C01839=1169.339,155.960,-56.654,-178.409,6.633,148.750
C01840=1169.335,156.209,-56.676,-178.406,6.635,148.750
C01841=1169.329,156.458,-56.697,-178.404,6.637,148.750
C01842=1169.325,156.707,-56.718,-178.401,6.639,148.749
C01843=1169.321,156.956,-56.739,-178.398,6.640,148.749
C01844=1169.316,157.205,-56.761,-178.396,6.642,148.748
C01845=1169.311,157.454,-56.783,-178.393,6.644,148.748
C01846=1169.306,157.703,-56.803,-178.390,6.646,148.748
C01847=1169.301,157.972,-56.828,-178.388,6.647,148.747
C01848=1169.296,158.241,-56.850,-178.384,6.650,148.747
C01849=1169.290,158.510,-56.874,-178.382,6.652,148.747
C01850=1169.286,158.779,-56.896,-178.378,6.653,148.746
C01851=1169.281,159.028,-56.918,-178.376,6.655,148.746
C01852=1169.276,159.277,-56.940,-178.374,6.657,148.745
C01853=1169.272,159.526,-56.962,-178.370,6.659,148.745
C01854=1169.266,159.775,-56.983,-178.368,6.661,148.745
C01855=1169.262,160.024,-57.005,-178.365,6.663,148.744
C01856=1169.257,160.273,-57.027,-178.362,6.665,148.744
C01857=1169.253,160.522,-57.049,-178.360,6.666,148.744
C01858=1169.248,160.772,-57.070,-178.357,6.668,148.743
C01859=1169.243,161.020,-57.091,-178.354,6.670,148.743
C01860=1169.239,161.270,-57.113,-178.351,6.672,148.742
C01861=1169.234,161.518,-57.135,-178.349,6.673,148.742
C01862=1169.229,161.767,-57.157,-178.346,6.675,148.742
C01863=1169.225,162.016,-57.179,-178.343,6.677,148.741
C01864=1169.220,162.266,-57.200,-178.341,6.679,148.741
C01865=1169.215,162.515,-57.222,-178.338,6.680,148.741
C01866=1169.210,162.764,-57.243,-178.335,6.682,148.740
C01867=1169.206,163.012,-57.265,-178.332,6.685,148.740
C01868=1169.201,163.261,-57.287,-178.329,6.687,148.739
C01869=1169.196,163.510,-57.309,-178.327,6.688,148.739
C01870=1169.192,163.759,-57.331,-178.324,6.690,148.739
C01871=1169.187,164.008,-57.353,-178.322,6.692,148.739
C01872=1169.183,164.257,-57.375,-178.319,6.694,148.738
C01873=1169.178,164.506,-57.396,-178.316,6.696,148.738
C01874=1169.173,164.755,-57.418,-178.314,6.697,148.737
C01875=1169.169,165.004,-57.440,-178.311,6.699,148.737
C01876=1169.164,165.253,-57.462,-178.308,6.701,148.737
C01877=1169.160,165.502,-57.484,-178.306,6.703,148.736
C01878=1169.155,165.751,-57.505,-178.302,6.705,148.736
C01879=1169.150,166.000,-57.528,-178.300,6.707,148.736
C01880=1169.145,166.249,-57.550,-178.297,6.709,148.735
C01881=1169.141,166.498,-57.572,-178.294,6.711,148.735
C01882=1169.136,166.747,-57.593,-178.292,6.712,148.735
C01883=1169.132,166.996,-57.616,-178.289,6.714,148.734
C01884=1169.127,167.245,-57.637,-178.287,6.716,148.734
C01885=1169.123,167.494,-57.659,-178.284,6.718,148.734
C01886=1169.117,167.743,-57.682,-178.281,6.720,148.733
C01887=1169.113,167.993,-57.704,-178.278,6.722,148.733
C01888=1169.108,168.241,-57.725,-178.275,6.724,148.733
C01889=1169.104,168.490,-57.748,-178.273,6.726,148.732
C01890=1169.099,168.739,-57.770,-178.270,6.728,148.732
C01891=1169.094,168.988,-57.792,-178.267,6.729,148.731
C01892=1169.089,169.237,-57.814,-178.265,6.731,148.731
C01893=1169.085,169.486,-57.836,-178.262,6.733,148.731
C01894=1169.080,169.735,-57.858,-178.260,6.735,148.731
C01895=1169.075,169.984,-57.881,-178.257,6.737,148.730
C01896=1169.070,170.233,-57.903,-178.254,6.739,148.730
C01897=1169.066,170.482,-57.925,-178.251,6.741,148.729
C01898=1169.062,170.731,-57.947,-178.248,6.743,148.729
C01899=1169.057,170.980,-57.970,-178.246,6.745,148.729
C01900=1169.052,171.229,-57.992,-178.243,6.746,148.728
C01901=1169.047,171.478,-58.014,-178.240,6.748,148.728
C01902=1169.042,171.727,-58.036,-178.238,6.751,148.728
C01903=1169.038,171.975,-58.059,-178.235,6.753,148.728
C01904=1169.034,172.225,-58.081,-178.232,6.754,148.727
C01905=1169.029,172.474,-58.103,-178.230,6.756,148.727
C01906=1169.024,172.722,-58.126,-178.227,6.758,148.726
C01907=1169.020,172.972,-58.148,-178.224,6.760,148.726
C01908=1169.014,173.221,-58.170,-178.221,6.762,148.726
C01909=1169.010,173.469,-58.193,-178.218,6.764,148.725
C01910=1169.006,173.719,-58.215,-178.216,6.766,148.725
C01911=1169.000,173.968,-58.237,-178.213,6.768,148.725
C01912=1168.996,174.216,-58.260,-178.211,6.770,148.724
C01913=1168.991,174.465,-58.282,-178.208,6.771,148.724
C01914=1168.987,174.714,-58.305,-178.205,6.774,148.724
C01915=1168.983,174.963,-58.327,-178.202,6.776,148.723
C01916=1168.977,175.212,-58.350,-178.199,6.778,148.723
C01917=1168.973,175.461,-58.372,-178.197,6.780,148.723
C01918=1168.968,175.711,-58.395,-178.194,6.781,148.723
C01919=1168.963,175.959,-58.417,-178.192,6.783,148.722
C01920=1168.959,176.208,-58.439,-178.188,6.786,148.722
C01921=1168.954,176.457,-58.463,-178.186,6.788,148.721
C01922=1168.950,176.706,-58.484,-178.183,6.789,148.721
C01923=1168.945,176.955,-58.508,-178.181,6.791,148.721
C01924=1168.941,177.203,-58.530,-178.178,6.793,148.721
C01925=1168.935,177.452,-58.553,-178.176,6.795,148.720
C01926=1168.931,177.701,-58.575,-178.172,6.798,148.720
C01927=1168.926,177.951,-58.598,-178.170,6.799,148.720
C01928=1168.922,178.199,-58.621,-178.167,6.801,148.719
C01929=1168.917,178.448,-58.643,-178.165,6.803,148.719
C01930=1168.913,178.697,-58.666,-178.162,6.805,148.719
C01931=1168.908,178.946,-58.689,-178.159,6.808,148.718
C01932=1168.903,179.195,-58.711,-178.156,6.809,148.718
C01933=1168.898,179.444,-58.734,-178.153,6.811,148.718
C01934=1168.895,179.693,-58.757,-178.151,6.813,148.717
C01935=1168.890,179.942,-58.780,-178.149,6.815,148.717
C01936=1168.885,180.190,-58.802,-178.145,6.818,148.717
C01937=1168.880,180.439,-58.825,-178.143,6.819,148.716
C01938=1168.875,180.689,-58.848,-178.140,6.821,148.716
C01939=1168.871,180.938,-58.871,-178.137,6.823,148.716
C01940=1168.866,181.186,-58.894,-178.134,6.826,148.716
C01941=1168.862,181.435,-58.916,-178.132,6.827,148.715
C01942=1168.857,181.684,-58.939,-178.129,6.829,148.715
C01943=1168.852,181.933,-58.963,-178.126,6.831,148.714
C01944=1168.848,182.182,-58.985,-178.124,6.833,148.714
C01945=1168.843,182.430,-59.008,-178.121,6.836,148.714
C01946=1168.839,182.680,-59.030,-178.118,6.837,148.714
C01947=1168.834,182.929,-59.054,-178.116,6.839,148.713
C01948=1168.829,183.178,-59.077,-178.113,6.841,148.713
C01949=1168.825,183.427,-59.100,-178.110,6.844,148.713
C01950=1168.820,183.675,-59.123,-178.107,6.846,148.712
C01951=1168.815,183.945,-59.148,-178.105,6.847,148.712
C01952=1168.810,184.214,-59.172,-178.101,6.850,148.712
C01953=1168.806,184.485,-59.198,-178.099,6.852,148.711
C01954=1168.800,184.754,-59.223,-178.096,6.854,148.711
C01955=1168.796,185.002,-59.245,-178.093,6.856,148.711
C01956=1168.791,185.251,-59.268,-178.091,6.858,148.711
C01957=1168.786,185.500,-59.292,-178.087,6.861,148.710
C01958=1168.782,185.749,-59.315,-178.085,6.863,148.710
C01959=1168.778,185.998,-59.338,-178.082,6.864,148.710
C01960=1168.773,186.247,-59.361,-178.079,6.866,148.709
C01961=1168.768,186.496,-59.385,-178.077,6.869,148.709
C01962=1168.763,186.745,-59.408,-178.074,6.871,148.709
C01963=1168.759,186.993,-59.430,-178.071,6.873,148.708
C01964=1168.754,187.242,-59.454,-178.069,6.874,148.708
C01965=1168.750,187.491,-59.477,-178.066,6.877,148.708
C01966=1168.745,187.740,-59.501,-178.063,6.879,148.708
C01967=1168.740,187.989,-59.524,-178.060,6.881,148.707
C01968=1168.736,188.238,-59.547,-178.058,6.883,148.707
C01969=1168.731,188.487,-59.570,-178.055,6.886,148.707
C01970=1168.727,188.736,-59.593,-178.052,6.887,148.706
C01971=1168.722,188.985,-59.617,-178.050,6.889,148.706
C01972=1168.717,189.234,-59.640,-178.047,6.891,148.706
C01973=1168.712,189.483,-59.663,-178.044,6.894,148.706
C01974=1168.707,189.732,-59.686,-178.041,6.896,148.705
C01975=1168.704,189.980,-59.710,-178.039,6.897,148.705
C01976=1168.699,190.229,-59.733,-178.036,6.900,148.705
C01977=1168.694,190.478,-59.757,-178.033,6.902,148.704
C01978=1168.690,190.727,-59.780,-178.031,6.904,148.704
C01979=1168.685,190.976,-59.803,-178.028,6.906,148.704
C01980=1168.680,191.225,-59.827,-178.025,6.909,148.704
C01981=1168.676,191.473,-59.851,-178.023,6.910,148.703
C01982=1168.671,191.722,-59.874,-178.020,6.912,148.703
C01983=1168.666,191.971,-59.897,-178.017,6.915,148.703
C01984=1168.662,192.220,-59.921,-178.014,6.917,148.702
C01985=1168.657,192.469,-59.945,-178.012,6.919,148.702
C01986=1168.653,192.718,-59.968,-178.009,6.920,148.702
C01987=1168.648,192.967,-59.992,-178.006,6.923,148.702
C01988=1168.643,193.216,-60.015,-178.004,6.925,148.701
C01989=1168.639,193.464,-60.039,-178.001,6.927,148.701
C01990=1168.634,193.713,-60.062,-177.998,6.929,148.701
C01991=1168.629,193.962,-60.086,-177.995,6.932,148.700
C01992=1168.625,194.211,-60.110,-177.993,6.933,148.700
C01993=1168.620,194.460,-60.133,-177.990,6.936,148.700
C01994=1168.616,194.709,-60.157,-177.987,6.938,148.700
C01995=1168.611,194.957,-60.181,-177.985,6.940,148.699
C01996=1168.607,195.206,-60.204,-177.981,6.942,148.699
C01997=1168.602,195.455,-60.228,-177.979,6.945,148.699
C01998=1168.597,195.704,-60.251,-177.977,6.946,148.698
C01999=1168.593,195.953,-60.275,-177.974,6.948,148.698
C02000=1168.588,196.201,-60.299,-177.971,6.951,148.698
C02001=1168.584,196.450,-60.322,-177.968,6.953,148.698
C02002=1168.579,196.699,-60.346,-177.966,6.955,148.697
C02003=1168.575,196.948,-60.370,-177.963,6.957,148.697
C02004=1168.571,197.197,-60.394,-177.960,6.959,148.697
C02005=1168.566,197.446,-60.417,-177.958,6.961,148.696
C02006=1168.561,197.695,-60.442,-177.955,6.964,148.696
C02007=1168.556,197.944,-60.466,-177.952,6.966,148.696
C02008=1168.552,198.192,-60.490,-177.950,6.968,148.696
C02009=1168.547,198.441,-60.513,-177.947,6.970,148.696
C02010=1168.543,198.689,-60.537,-177.944,6.972,148.695
C02011=1168.538,198.938,-60.560,-177.941,6.974,148.695
C02012=1168.534,199.187,-60.584,-177.939,6.977,148.695
C02013=1168.529,199.436,-60.609,-177.936,6.979,148.694
C02014=1168.524,199.685,-60.633,-177.933,6.981,148.694
C02015=1168.520,199.934,-60.657,-177.930,6.983,148.694
C02016=1168.515,200.183,-60.680,-177.928,6.985,148.694
C02017=1168.511,200.431,-60.704,-177.925,6.988,148.693
C02018=1168.507,200.680,-60.728,-177.922,6.990,148.693
C02019=1168.501,200.929,-60.752,-177.920,6.992,148.693
C02020=1168.497,201.178,-60.777,-177.916,6.994,148.692
C02021=1168.493,201.426,-60.801,-177.914,6.996,148.692
C02022=1168.488,201.675,-60.824,-177.912,6.998,148.692
C02023=1168.483,201.924,-60.849,-177.908,7.001,148.692
C02024=1168.479,202.173,-60.873,-177.906,7.003,148.692
C02025=1168.474,202.421,-60.897,-177.903,7.005,148.691
C02026=1168.470,202.671,-60.921,-177.901,7.008,148.691
C02027=1168.465,202.919,-60.945,-177.898,7.009,148.691
C02028=1168.461,203.168,-60.970,-177.895,7.012,148.690
C02029=1168.456,203.416,-60.994,-177.893,7.014,148.690
C02030=1168.451,203.666,-61.018,-177.890,7.016,148.690
C02031=1168.447,203.915,-61.042,-177.887,7.018,148.690
C02032=1168.443,204.163,-61.066,-177.884,7.021,148.690
C02033=1168.438,204.412,-61.091,-177.882,7.022,148.689
C02034=1168.433,204.660,-61.115,-177.879,7.025,148.689
C02035=1168.429,204.909,-61.139,-177.876,7.027,148.689
C02036=1168.424,205.159,-61.163,-177.873,7.030,148.688
C02037=1168.419,205.407,-61.187,-177.871,7.032,148.688
C02038=1168.415,205.656,-61.211,-177.868,7.034,148.688
C02039=1168.411,205.905,-61.236,-177.865,7.037,148.688
C02040=1168.406,206.153,-61.260,-177.863,7.038,148.688
C02041=1168.401,206.402,-61.285,-177.860,7.041,148.687
C02042=1168.397,206.651,-61.309,-177.857,7.043,148.687
C02043=1168.393,206.900,-61.334,-177.855,7.045,148.687
C02044=1168.388,207.148,-61.358,-177.852,7.048,148.687
C02045=1168.383,207.397,-61.382,-177.849,7.050,148.686
C02046=1168.379,207.646,-61.407,-177.846,7.052,148.686
C02047=1168.374,207.895,-61.432,-177.844,7.054,148.686
C02048=1168.369,208.143,-61.456,-177.841,7.056,148.686
C02049=1168.365,208.392,-61.480,-177.838,7.059,148.685
C02050=1168.360,208.641,-61.505,-177.836,7.061,148.685
C02051=1168.356,208.890,-61.529,-177.832,7.063,148.685
C02052=1168.351,209.138,-61.554,-177.830,7.065,148.685
C02053=1168.347,209.387,-61.578,-177.827,7.068,148.684
C02054=1168.342,209.636,-61.603,-177.825,7.070,148.684
C02055=1168.337,209.906,-61.629,-177.822,7.073,148.684
C02056=1168.333,210.177,-61.656,-177.819,7.075,148.684
C02057=1168.328,210.447,-61.683,-177.816,7.078,148.683
C02058=1168.323,210.717,-61.710,-177.813,7.080,148.683
C02059=1168.318,210.967,-61.735,-177.810,7.082,148.683
C02060=1168.314,211.215,-61.759,-177.807,7.085,148.683
C02061=1168.309,211.465,-61.784,-177.805,7.087,148.682
C02062=1168.304,211.713,-61.809,-177.802,7.090,148.682
C02063=1168.300,211.962,-61.833,-177.799,7.091,148.682
C02064=1168.295,212.210,-61.858,-177.797,7.094,148.682
C02065=1168.291,212.459,-61.882,-177.794,7.096,148.681
C02066=1168.286,212.708,-61.908,-177.792,7.098,148.681
C02067=1168.281,212.957,-61.932,-177.788,7.101,148.681
C02068=1168.277,213.205,-61.957,-177.786,7.103,148.681
C02069=1168.273,213.454,-61.982,-177.783,7.106,148.681
C02070=1168.268,213.703,-62.006,-177.780,7.107,148.680
C02071=1168.264,213.952,-62.031,-177.778,7.110,148.680
C02072=1168.259,214.200,-62.057,-177.775,7.112,148.680
C02073=1168.255,214.449,-62.081,-177.773,7.114,148.680
C02074=1168.250,214.698,-62.106,-177.769,7.117,148.679
C02075=1168.245,214.946,-62.131,-177.767,7.119,148.679
C02076=1168.241,215.195,-62.155,-177.764,7.122,148.679
C02077=1168.236,215.444,-62.180,-177.762,7.124,148.679
C02078=1168.232,215.693,-62.206,-177.759,7.126,148.679
C02079=1168.228,215.941,-62.230,-177.756,7.128,148.678
C02080=1168.223,216.190,-62.256,-177.753,7.131,148.678
C02081=1168.218,216.439,-62.280,-177.751,7.133,148.678
C02082=1168.214,216.688,-62.305,-177.748,7.136,148.678
C02083=1168.210,216.936,-62.330,-177.746,7.138,148.678
C02084=1168.205,217.185,-62.355,-177.742,7.140,148.677
C02085=1168.200,217.433,-62.381,-177.740,7.143,148.677
C02086=1168.195,217.682,-62.405,-177.737,7.145,148.677
C02087=1168.192,217.931,-62.430,-177.735,7.147,148.677
C02088=1168.187,218.179,-62.455,-177.731,7.150,148.676
C02089=1168.182,218.428,-62.481,-177.729,7.152,148.676
C02090=1168.178,218.678,-62.506,-177.727,7.154,148.676
C02091=1168.173,218.926,-62.531,-177.724,7.157,148.676
C02092=1168.169,219.175,-62.556,-177.721,7.159,148.676
C02093=1168.164,219.423,-62.581,-177.718,7.161,148.675
C02094=1168.160,219.672,-62.607,-177.716,7.163,148.675
C02095=1168.155,219.920,-62.632,-177.713,7.166,148.675
C02096=1168.151,220.169,-62.657,-177.710,7.168,148.675
C02097=1168.146,220.418,-62.681,-177.708,7.171,148.675
C02098=1168.142,220.666,-62.707,-177.705,7.173,148.674
C02099=1168.137,220.915,-62.732,-177.702,7.176,148.674
C02100=1168.133,221.164,-62.758,-177.699,7.177,148.674
C02101=1168.129,221.413,-62.783,-177.697,7.180,148.674
C02102=1168.124,221.661,-62.809,-177.694,7.182,148.673
C02103=1168.119,221.910,-62.834,-177.691,7.185,148.673
C02104=1168.114,222.158,-62.859,-177.688,7.188,148.673
C02105=1168.110,222.407,-62.885,-177.686,7.190,148.673
C02106=1168.106,222.656,-62.909,-177.683,7.193,148.673
C02107=1168.102,222.904,-62.935,-177.680,7.195,148.673
C02108=1168.097,223.153,-62.960,-177.678,7.198,148.672
C02109=1168.093,223.401,-62.986,-177.675,7.199,148.672
C02110=1168.088,223.651,-63.011,-177.672,7.202,148.672
C02111=1168.084,223.900,-63.037,-177.670,7.204,148.672
C02112=1168.079,224.148,-63.062,-177.667,7.207,148.672
C02113=1168.075,224.397,-63.088,-177.664,7.209,148.671
C02114=1168.070,224.645,-63.113,-177.661,7.212,148.671
C02115=1168.065,224.894,-63.138,-177.659,7.214,148.671
C02116=1168.061,225.143,-63.164,-177.656,7.217,148.671
C02117=1168.056,225.391,-63.189,-177.654,7.219,148.671
C02118=1168.052,225.640,-63.215,-177.650,7.221,148.670
C02119=1168.048,225.889,-63.241,-177.648,7.223,148.670
C02120=1168.043,226.137,-63.266,-177.645,7.226,148.670
C02121=1168.039,226.385,-63.292,-177.642,7.229,148.670
C02122=1168.035,226.634,-63.318,-177.640,7.231,148.670
C02123=1168.030,226.882,-63.343,-177.637,7.234,148.669
C02124=1168.025,227.132,-63.369,-177.635,7.236,148.669
C02125=1168.020,227.381,-63.394,-177.631,7.238,148.669
C02126=1168.015,227.629,-63.420,-177.629,7.241,148.669
C02127=1168.011,227.878,-63.446,-177.626,7.243,148.669
C02128=1168.007,228.127,-63.471,-177.624,7.245,148.669
C02129=1168.003,228.375,-63.497,-177.621,7.248,148.668
C02130=1167.998,228.624,-63.522,-177.618,7.251,148.668
C02131=1167.994,228.872,-63.548,-177.616,7.253,148.668
C02132=1167.990,229.121,-63.574,-177.612,7.256,148.668
C02133=1167.985,229.370,-63.601,-177.610,7.258,148.668
C02134=1167.980,229.618,-63.626,-177.607,7.261,148.668
C02135=1167.976,229.867,-63.652,-177.605,7.262,148.667
C02136=1167.972,230.115,-63.678,-177.602,7.265,148.667
C02137=1167.967,230.364,-63.704,-177.599,7.268,148.667
C02138=1167.963,230.612,-63.729,-177.597,7.270,148.667
C02139=1167.958,230.861,-63.755,-177.594,7.273,148.667
C02140=1167.953,231.110,-63.781,-177.591,7.275,148.666
C02141=1167.949,231.359,-63.807,-177.588,7.278,148.666
C02142=1167.945,231.606,-63.833,-177.586,7.280,148.666
C02143=1167.940,231.856,-63.859,-177.583,7.283,148.666
C02144=1167.935,232.104,-63.885,-177.580,7.286,148.666
C02145=1167.931,232.353,-63.911,-177.578,7.287,148.665
C02146=1167.927,232.602,-63.937,-177.575,7.290,148.665
C02147=1167.922,232.850,-63.963,-177.573,7.292,148.665
C02148=1167.917,233.099,-63.989,-177.569,7.295,148.665
C02149=1167.913,233.347,-64.015,-177.567,7.298,148.665
C02150=1167.909,233.596,-64.041,-177.564,7.300,148.665
C02151=1167.904,233.845,-64.068,-177.561,7.303,148.664
C02152=1167.900,234.093,-64.093,-177.559,7.305,148.664
C02153=1167.895,234.342,-64.119,-177.556,7.308,148.664
C02154=1167.891,234.590,-64.146,-177.553,7.310,148.664
C02155=1167.886,234.839,-64.172,-177.551,7.313,148.664
C02156=1167.882,235.088,-64.197,-177.548,7.316,148.664
C02157=1167.878,235.336,-64.224,-177.545,7.317,148.663
C02158=1167.873,235.585,-64.250,-177.543,7.320,148.663
C02159=1167.868,235.856,-64.278,-177.539,7.323,148.663
C02160=1167.863,236.128,-64.307,-177.537,7.326,148.663
C02161=1167.859,236.399,-64.336,-177.534,7.329,148.663
C02162=1167.853,236.671,-64.365,-177.531,7.331,148.663
C02163=1167.849,236.919,-64.391,-177.528,7.334,148.663
C02164=1167.845,237.168,-64.417,-177.526,7.336,148.663
C02165=1167.840,237.417,-64.444,-177.523,7.339,148.662
C02166=1167.836,237.666,-64.470,-177.520,7.341,148.662
C02167=1167.831,237.914,-64.497,-177.518,7.344,148.662
C02168=1167.827,238.163,-64.522,-177.514,7.347,148.662
C02169=1167.823,238.411,-64.549,-177.512,7.349,148.662
C02170=1167.818,238.660,-64.575,-177.509,7.352,148.662
C02171=1167.814,238.908,-64.601,-177.506,7.355,148.661
C02172=1167.809,239.157,-64.628,-177.504,7.357,148.661
C02173=1167.805,239.405,-64.654,-177.501,7.360,148.661
C02174=1167.800,239.654,-64.680,-177.498,7.363,148.661
C02175=1167.796,239.902,-64.707,-177.496,7.364,148.661
C02176=1167.791,240.151,-64.734,-177.493,7.367,148.661
C02177=1167.787,240.400,-64.760,-177.490,7.370,148.661
C02178=1167.782,240.648,-64.787,-177.488,7.372,148.660
C02179=1167.778,240.897,-64.813,-177.485,7.375,148.660
C02180=1167.774,241.145,-64.840,-177.483,7.377,148.660
C02181=1167.769,241.394,-64.867,-177.480,7.380,148.660
C02182=1167.765,241.643,-64.892,-177.477,7.383,148.660
C02183=1167.760,241.891,-64.919,-177.474,7.385,148.660
C02184=1167.756,242.139,-64.946,-177.472,7.388,148.660
C02185=1167.752,242.388,-64.973,-177.469,7.391,148.659
C02186=1167.747,242.637,-64.999,-177.466,7.393,148.659
C02187=1167.743,242.885,-65.026,-177.464,7.395,148.659
C02188=1167.738,243.134,-65.053,-177.461,7.398,148.659
C02189=1167.734,243.382,-65.079,-177.459,7.401,148.659
C02190=1167.729,243.631,-65.106,-177.455,7.403,148.659
C02191=1167.725,243.879,-65.132,-177.453,7.406,148.659
C02192=1167.721,244.128,-65.159,-177.450,7.409,148.658
C02193=1167.716,244.376,-65.186,-177.448,7.411,148.658
C02194=1167.712,244.624,-65.213,-177.444,7.414,148.658
C02195=1167.707,244.873,-65.239,-177.442,7.417,148.658
C02196=1167.702,245.122,-65.266,-177.440,7.419,148.658
C02197=1167.698,245.370,-65.293,-177.437,7.422,148.658
C02198=1167.694,245.619,-65.320,-177.434,7.425,148.658
C02199=1167.690,245.868,-65.347,-177.431,7.427,148.657
C02200=1167.685,246.116,-65.374,-177.429,7.430,148.657
C02201=1167.681,246.364,-65.401,-177.426,7.433,148.657
C02202=1167.676,246.613,-65.428,-177.424,7.435,148.657
C02203=1167.672,246.861,-65.455,-177.420,7.437,148.657
C02204=1167.668,247.110,-65.481,-177.418,7.440,148.657
C02205=1167.663,247.358,-65.508,-177.415,7.442,148.657
C02206=1167.659,247.607,-65.535,-177.413,7.445,148.657
C02207=1167.654,247.855,-65.562,-177.410,7.448,148.657
C02208=1167.650,248.103,-65.589,-177.407,7.451,148.656
C02209=1167.646,248.353,-65.616,-177.405,7.453,148.656
C02210=1167.641,248.601,-65.643,-177.402,7.456,148.656
C02211=1167.637,248.850,-65.670,-177.399,7.459,148.656
C02212=1167.632,249.098,-65.697,-177.397,7.461,148.656
C02213=1167.628,249.346,-65.724,-177.394,7.464,148.656
C02214=1167.623,249.595,-65.751,-177.391,7.467,148.656
C02215=1167.619,249.843,-65.778,-177.388,7.470,148.656
C02216=1167.615,250.092,-65.805,-177.386,7.472,148.656
C02217=1167.610,250.341,-65.833,-177.383,7.475,148.655
C02218=1167.605,250.589,-65.860,-177.380,7.478,148.655
C02219=1167.601,250.838,-65.887,-177.378,7.480,148.655
C02220=1167.597,251.085,-65.914,-177.375,7.482,148.655
C02221=1167.593,251.335,-65.941,-177.372,7.485,148.655
C02222=1167.588,251.583,-65.968,-177.369,7.488,148.655
C02223=1167.584,251.832,-65.995,-177.367,7.491,148.655
C02224=1167.579,252.080,-66.022,-177.365,7.493,148.655
C02225=1167.575,252.328,-66.050,-177.362,7.496,148.655
C02226=1167.571,252.577,-66.078,-177.359,7.499,148.654
C02227=1167.566,252.826,-66.105,-177.356,7.501,148.654
C02228=1167.561,253.074,-66.132,-177.354,7.504,148.654
C02229=1167.557,253.322,-66.160,-177.351,7.507,148.654
C02230=1167.552,253.571,-66.187,-177.348,7.510,148.654
C02231=1167.548,253.820,-66.214,-177.346,7.512,148.654
C02232=1167.544,254.068,-66.242,-177.343,7.515,148.654
C02233=1167.540,254.316,-66.268,-177.340,7.518,148.654
C02234=1167.535,254.564,-66.295,-177.337,7.521,148.654
C02235=1167.532,254.813,-66.323,-177.335,7.523,148.654
C02236=1167.527,255.061,-66.351,-177.332,7.526,148.653
C02237=1167.522,255.310,-66.378,-177.330,7.529,148.653
C02238=1167.517,255.558,-66.406,-177.327,7.532,148.653
C02239=1167.513,255.807,-66.433,-177.325,7.534,148.653
C02240=1167.509,256.055,-66.461,-177.322,7.537,148.653
C02241=1167.504,256.304,-66.488,-177.319,7.540,148.653
C02242=1167.500,256.552,-66.516,-177.316,7.542,148.653
C02243=1167.496,256.801,-66.543,-177.314,7.545,148.653
C02244=1167.491,257.049,-66.571,-177.311,7.548,148.653
C02245=1167.487,257.298,-66.599,-177.308,7.551,148.653
C02246=1167.483,257.546,-66.626,-177.305,7.553,148.653
C02247=1167.478,257.794,-66.653,-177.303,7.556,148.652
C02248=1167.474,258.043,-66.681,-177.300,7.559,148.652
C02249=1167.470,258.291,-66.709,-177.298,7.562,148.652
C02250=1167.465,258.539,-66.737,-177.295,7.564,148.652
C02251=1167.461,258.789,-66.765,-177.292,7.567,148.652
C02252=1167.456,259.036,-66.792,-177.290,7.570,148.652
C02253=1167.452,259.285,-66.819,-177.287,7.572,148.652
C02254=1167.448,259.534,-66.847,-177.284,7.575,148.652
C02255=1167.444,259.781,-66.875,-177.281,7.578,148.652
C02256=1167.439,260.030,-66.902,-177.279,7.580,148.652
C02257=1167.435,260.279,-66.931,-177.276,7.583,148.652
C02258=1167.430,260.527,-66.958,-177.274,7.586,148.652
C02259=1167.426,260.775,-66.986,-177.271,7.589,148.651
C02260=1167.422,261.024,-67.014,-177.268,7.592,148.651
C02261=1167.417,261.272,-67.042,-177.266,7.594,148.651
C02262=1167.413,261.521,-67.070,-177.263,7.597,148.651
C02263=1167.407,261.794,-67.100,-177.260,7.600,148.651
C02264=1167.403,262.067,-67.131,-177.257,7.604,148.651
C02265=1167.398,262.340,-67.162,-177.254,7.607,148.651
C02266=1167.394,262.613,-67.193,-177.251,7.610,148.651
C02267=1167.389,262.862,-67.220,-177.248,7.612,148.651
C02268=1167.385,263.110,-67.248,-177.246,7.615,148.651
C02269=1167.380,263.358,-67.276,-177.243,7.618,148.651
C02270=1167.376,263.606,-67.304,-177.241,7.621,148.651
C02271=1167.372,263.855,-67.332,-177.238,7.624,148.651
C02272=1167.367,264.104,-67.360,-177.235,7.626,148.651
C02273=1167.363,264.352,-67.388,-177.232,7.629,148.650
C02274=1167.359,264.600,-67.416,-177.230,7.632,148.650
C02275=1167.354,264.849,-67.445,-177.227,7.635,148.650
C02276=1167.350,265.097,-67.472,-177.225,7.638,148.650
C02277=1167.346,265.345,-67.501,-177.222,7.640,148.650
C02278=1167.341,265.594,-67.529,-177.219,7.643,148.650
C02279=1167.337,265.842,-67.557,-177.217,7.646,148.650
C02280=1167.333,266.090,-67.585,-177.214,7.649,148.650
C02281=1167.328,266.339,-67.614,-177.212,7.651,148.650
C02282=1167.324,266.587,-67.641,-177.209,7.654,148.650
C02283=1167.319,266.836,-67.670,-177.206,7.657,148.650
C02284=1167.315,267.084,-67.698,-177.203,7.660,148.650
C02285=1167.311,267.332,-67.726,-177.201,7.663,148.650
C02286=1167.306,267.580,-67.754,-177.198,7.665,148.650
C02287=1167.303,267.829,-67.783,-177.196,7.668,148.650
C02288=1167.297,268.077,-67.811,-177.193,7.671,148.650
C02289=1167.294,268.326,-67.839,-177.190,7.674,148.650
C02290=1167.289,268.574,-67.867,-177.187,7.677,148.649
C02291=1167.285,268.822,-67.896,-177.185,7.679,148.649
C02292=1167.280,269.071,-67.924,-177.182,7.682,148.649
C02293=1167.276,269.319,-67.952,-177.180,7.686,148.650
C02294=1167.272,269.568,-67.981,-177.177,7.689,148.649
C02295=1167.267,269.816,-68.009,-177.175,7.692,148.649
C02296=1167.263,270.065,-68.037,-177.172,7.695,148.649
C02297=1167.259,270.312,-68.066,-177.169,7.698,148.649
C02298=1167.254,270.561,-68.095,-177.167,7.700,148.649
C02299=1167.250,270.809,-68.122,-177.164,7.703,148.649
C02300=1167.245,271.058,-68.151,-177.161,7.706,148.649
C02301=1167.242,271.306,-68.179,-177.159,7.709,148.649
C02302=1167.237,271.554,-68.208,-177.156,7.712,148.649
C02303=1167.232,271.803,-68.237,-177.153,7.715,148.649
C02304=1167.228,272.051,-68.265,-177.150,7.717,148.649
C02305=1167.223,272.300,-68.294,-177.148,7.720,148.649
C02306=1167.220,272.548,-68.322,-177.145,7.723,148.649
C02307=1167.215,272.796,-68.351,-177.143,7.726,148.649
C02308=1167.210,273.045,-68.380,-177.140,7.729,148.649
C02309=1167.207,273.293,-68.408,-177.138,7.732,148.649
C02310=1167.202,273.541,-68.437,-177.135,7.735,148.649
C02311=1167.197,273.790,-68.466,-177.132,7.738,148.649
C02312=1167.194,274.038,-68.494,-177.130,7.740,148.649
C02313=1167.189,274.286,-68.523,-177.127,7.743,148.649
C02314=1167.185,274.534,-68.552,-177.124,7.746,148.649
C02315=1167.181,274.783,-68.580,-177.122,7.749,148.649
C02316=1167.176,275.031,-68.609,-177.119,7.752,148.649
C02317=1167.172,275.279,-68.638,-177.116,7.755,148.648
C02318=1167.168,275.528,-68.666,-177.113,7.758,148.648
C02319=1167.163,275.775,-68.695,-177.111,7.761,148.649
C02320=1167.159,276.024,-68.724,-177.109,7.763,148.648
C02321=1167.155,276.272,-68.753,-177.106,7.766,148.648
C02322=1167.151,276.521,-68.782,-177.104,7.769,148.648
C02323=1167.146,276.769,-68.811,-177.101,7.772,148.648
C02324=1167.141,277.017,-68.840,-177.098,7.775,148.648
C02325=1167.138,277.265,-68.868,-177.095,7.778,148.648
C02326=1167.133,277.514,-68.897,-177.093,7.781,148.648
C02327=1167.129,277.762,-68.926,-177.090,7.784,148.648
C02328=1167.124,278.011,-68.955,-177.087,7.787,148.648
C02329=1167.120,278.259,-68.984,-177.085,7.789,148.648
C02330=1167.116,278.506,-69.013,-177.083,7.792,148.648
C02331=1167.112,278.755,-69.042,-177.080,7.795,148.648
C02332=1167.107,279.003,-69.071,-177.077,7.798,148.648
C02333=1167.103,279.252,-69.101,-177.074,7.801,148.648
C02334=1167.099,279.501,-69.129,-177.072,7.804,148.648
C02335=1167.095,279.748,-69.158,-177.069,7.807,148.648
C02336=1167.090,279.996,-69.187,-177.067,7.810,148.648
C02337=1167.086,280.245,-69.216,-177.064,7.813,148.648
C02338=1167.082,280.493,-69.245,-177.061,7.816,148.648
C02339=1167.078,280.741,-69.275,-177.058,7.819,148.648
C02340=1167.073,280.990,-69.303,-177.056,7.821,148.648
C02341=1167.068,281.238,-69.333,-177.054,7.825,148.648
C02342=1167.064,281.486,-69.362,-177.051,7.828,148.648
C02343=1167.060,281.734,-69.392,-177.048,7.831,148.648
C02344=1167.056,281.983,-69.421,-177.046,7.834,148.648
C02345=1167.051,282.231,-69.449,-177.043,7.837,148.648
C02346=1167.047,282.479,-69.478,-177.040,7.840,148.648
C02347=1167.043,282.727,-69.508,-177.038,7.843,148.648
C02348=1167.039,282.975,-69.537,-177.035,7.846,148.648
C02349=1167.035,283.224,-69.567,-177.032,7.849,148.648
C02350=1167.031,283.472,-69.596,-177.030,7.852,148.648
C02351=1167.025,283.720,-69.625,-177.027,7.855,148.648
C02352=1167.021,283.968,-69.654,-177.024,7.858,148.648
C02353=1167.017,284.217,-69.683,-177.022,7.860,148.648
C02354=1167.013,284.465,-69.713,-177.020,7.863,148.648
C02355=1167.009,284.713,-69.742,-177.017,7.866,148.648
C02356=1167.005,284.961,-69.772,-177.014,7.869,148.648
C02357=1167.000,285.210,-69.801,-177.012,7.872,148.648
C02358=1166.996,285.458,-69.831,-177.009,7.875,148.648
C02359=1166.991,285.707,-69.861,-177.006,7.878,148.648
C02360=1166.986,285.954,-69.890,-177.004,7.881,148.648
C02361=1166.982,286.202,-69.919,-177.001,7.885,148.648
C02362=1166.978,286.451,-69.949,-176.998,7.887,148.648
C02363=1166.974,286.699,-69.978,-176.996,7.890,148.648
C02364=1166.970,286.947,-70.008,-176.993,7.893,148.648
C02365=1166.966,287.196,-70.037,-176.990,7.896,148.648
C02366=1166.961,287.444,-70.067,-176.988,7.900,148.648
C02367=1166.957,287.719,-70.100,-176.985,7.903,148.648
C02368=1166.952,287.994,-70.133,-176.982,7.906,148.648
C02369=1166.947,288.269,-70.166,-176.979,7.909,148.648
C02370=1166.942,288.543,-70.197,-176.976,7.912,148.648
C02371=1166.937,288.792,-70.228,-176.974,7.916,148.648
C02372=1166.933,289.040,-70.257,-176.971,7.919,148.648
C02373=1166.929,289.288,-70.287,-176.969,7.922,148.648
C02374=1166.925,289.536,-70.317,-176.966,7.925,148.648
C02375=1166.921,289.784,-70.346,-176.964,7.928,148.648
C02376=1166.916,290.033,-70.376,-176.961,7.931,148.648
C02377=1166.912,290.280,-70.406,-176.958,7.934,148.648
C02378=1166.908,290.529,-70.436,-176.955,7.937,148.648
C02379=1166.904,290.777,-70.465,-176.953,7.940,148.648
C02380=1166.900,291.025,-70.495,-176.950,7.943,148.648
C02381=1166.895,291.273,-70.525,-176.948,7.946,148.648
C02382=1166.891,291.521,-70.555,-176.945,7.949,148.648
C02383=1166.887,291.770,-70.585,-176.943,7.952,148.648
C02384=1166.883,292.018,-70.615,-176.940,7.955,148.648
C02385=1166.879,292.267,-70.645,-176.937,7.958,148.648
C02386=1166.874,292.515,-70.674,-176.935,7.961,148.649
C02387=1166.870,292.762,-70.704,-176.932,7.964,148.649
C02388=1166.866,293.011,-70.735,-176.929,7.967,148.649
C02389=1166.861,293.259,-70.764,-176.927,7.971,148.649
C02390=1166.857,293.507,-70.794,-176.924,7.974,148.649
C02391=1166.853,293.756,-70.824,-176.921,7.977,148.649
C02392=1166.849,294.003,-70.854,-176.919,7.980,148.649
C02393=1166.845,294.251,-70.884,-176.917,7.982,148.649
C02394=1166.840,294.499,-70.915,-176.914,7.985,148.649
C02395=1166.836,294.748,-70.944,-176.912,7.988,148.649
C02396=1166.832,294.995,-70.974,-176.909,7.991,148.649
C02397=1166.828,295.245,-71.005,-176.906,7.994,148.649
C02398=1166.824,295.492,-71.035,-176.904,7.997,148.649
C02399=1166.819,295.740,-71.064,-176.901,8.001,148.649
C02400=1166.815,295.988,-71.095,-176.899,8.004,148.649
C02401=1166.811,296.237,-71.124,-176.896,8.006,148.649
C02402=1166.806,296.485,-71.155,-176.894,8.010,148.649
C02403=1166.802,296.733,-71.185,-176.891,8.013,148.649
C02404=1166.798,296.982,-71.216,-176.888,8.016,148.649
C02405=1166.794,297.229,-71.246,-176.886,8.019,148.649
C02406=1166.790,297.478,-71.275,-176.883,8.022,148.649
C02407=1166.785,297.725,-71.306,-176.880,8.025,148.649
C02408=1166.781,297.974,-71.336,-176.878,8.028,148.649
C02409=1166.776,298.222,-71.366,-176.875,8.031,148.649
C02410=1166.773,298.469,-71.397,-176.873,8.034,148.649
C02411=1166.768,298.719,-71.427,-176.870,8.037,148.649
C02412=1166.764,298.966,-71.457,-176.868,8.040,148.649
C02413=1166.760,299.214,-71.488,-176.865,8.043,148.649
C02414=1166.756,299.462,-71.518,-176.863,8.047,148.650
C02415=1166.751,299.710,-71.548,-176.859,8.051,148.650
C02416=1166.747,299.959,-71.579,-176.857,8.054,148.650
C02417=1166.743,300.207,-71.609,-176.854,8.057,148.650
C02418=1166.738,300.455,-71.640,-176.851,8.060,148.650
C02419=1166.734,300.703,-71.670,-176.849,8.063,148.650
C02420=1166.730,300.951,-71.700,-176.846,8.066,148.650
C02421=1166.726,301.199,-71.731,-176.844,8.069,148.650
C02422=1166.722,301.447,-71.762,-176.841,8.072,148.650
C02423=1166.717,301.695,-71.792,-176.839,8.075,148.650
C02424=1166.713,301.943,-71.823,-176.836,8.079,148.650
C02425=1166.709,302.192,-71.854,-176.834,8.082,148.650
C02426=1166.704,302.440,-71.884,-176.831,8.084,148.650
C02427=1166.700,302.688,-71.914,-176.829,8.088,148.650
C02428=1166.696,302.936,-71.945,-176.826,8.091,148.650
C02429=1166.692,303.184,-71.976,-176.824,8.094,148.651
C02430=1166.688,303.432,-72.006,-176.821,8.097,148.650
C02431=1166.683,303.680,-72.037,-176.818,8.100,148.651
C02432=1166.679,303.928,-72.068,-176.816,8.103,148.651
C02433=1166.675,304.176,-72.098,-176.813,8.106,148.651
C02434=1166.671,304.424,-72.129,-176.811,8.110,148.651
C02435=1166.666,304.672,-72.160,-176.808,8.113,148.651
C02436=1166.663,304.921,-72.190,-176.806,8.116,148.651
C02437=1166.658,305.168,-72.221,-176.803,8.119,148.651
C02438=1166.654,305.416,-72.252,-176.800,8.122,148.651
C02439=1166.650,305.665,-72.283,-176.798,8.125,148.651
C02440=1166.646,305.913,-72.313,-176.795,8.128,148.651
C02441=1166.641,306.161,-72.344,-176.793,8.131,148.651
C02442=1166.637,306.409,-72.375,-176.790,8.134,148.651
C02443=1166.633,306.657,-72.406,-176.788,8.138,148.651
C02444=1166.628,306.905,-72.437,-176.785,8.141,148.651
C02445=1166.625,307.153,-72.468,-176.782,8.145,148.652
C02446=1166.620,307.401,-72.498,-176.779,8.148,148.652
C02447=1166.616,307.649,-72.529,-176.777,8.151,148.652
C02448=1166.612,307.898,-72.560,-176.774,8.154,148.652
C02449=1166.607,308.145,-72.592,-176.772,8.157,148.652
C02450=1166.603,308.393,-72.623,-176.769,8.160,148.652
C02451=1166.600,308.641,-72.653,-176.767,8.163,148.652
C02452=1166.595,308.889,-72.684,-176.764,8.166,148.652
C02453=1166.591,309.137,-72.716,-176.762,8.169,148.652
C02454=1166.587,309.385,-72.747,-176.759,8.173,148.652
C02455=1166.582,309.633,-72.777,-176.757,8.176,148.652
C02456=1166.578,309.882,-72.808,-176.754,8.179,148.652
C02457=1166.574,310.129,-72.840,-176.752,8.182,148.652
C02458=1166.570,310.378,-72.871,-176.749,8.185,148.653
C02459=1166.565,310.626,-72.902,-176.747,8.188,148.653
C02460=1166.561,310.873,-72.933,-176.744,8.192,148.653
C02461=1166.558,311.121,-72.964,-176.741,8.195,148.653
C02462=1166.553,311.369,-72.995,-176.739,8.199,148.653
C02463=1166.549,311.617,-73.026,-176.736,8.202,148.653
C02464=1166.545,311.865,-73.057,-176.734,8.205,148.653
C02465=1166.541,312.113,-73.089,-176.731,8.208,148.653
C02466=1166.536,312.361,-73.120,-176.729,8.211,148.653
C02467=1166.533,312.609,-73.152,-176.726,8.214,148.653
C02468=1166.528,312.857,-73.182,-176.724,8.217,148.654
C02469=1166.524,313.106,-73.214,-176.721,8.220,148.654
C02470=1166.520,313.353,-73.245,-176.719,8.224,148.654
C02471=1166.515,313.630,-73.280,-176.715,8.227,148.654
C02472=1166.510,313.908,-73.315,-176.712,8.232,148.654
C02473=1166.505,314.185,-73.350,-176.710,8.235,148.654
C02474=1166.501,314.462,-73.385,-176.707,8.239,148.654
C02475=1166.497,314.710,-73.417,-176.704,8.242,148.654
C02476=1166.493,314.958,-73.448,-176.702,8.245,148.654
C02477=1166.488,315.206,-73.480,-176.699,8.248,148.654
C02478=1166.484,315.454,-73.511,-176.697,8.251,148.655
C02479=1166.480,315.702,-73.543,-176.694,8.254,148.655
C02480=1166.476,315.949,-73.574,-176.692,8.257,148.655
C02481=1166.472,316.198,-73.605,-176.689,8.261,148.655
C02482=1166.467,316.445,-73.637,-176.687,8.264,148.655
C02483=1166.464,316.693,-73.669,-176.684,8.268,148.655
C02484=1166.459,316.941,-73.699,-176.681,8.271,148.655
C02485=1166.455,317.189,-73.731,-176.679,8.274,148.655
C02486=1166.451,317.438,-73.764,-176.676,8.277,148.656
C02487=1166.446,317.686,-73.794,-176.674,8.280,148.656
C02488=1166.442,317.934,-73.826,-176.671,8.284,148.656
C02489=1166.438,318.181,-73.858,-176.669,8.287,148.656
C02490=1166.434,318.429,-73.890,-176.666,8.290,148.656
C02491=1166.430,318.678,-73.921,-176.664,8.293,148.656
C02492=1166.425,318.925,-73.953,-176.661,8.297,148.656
C02493=1166.422,319.173,-73.985,-176.658,8.300,148.656
C02494=1166.417,319.421,-74.016,-176.656,8.303,148.656
C02495=1166.414,319.669,-74.048,-176.653,8.307,148.656
C02496=1166.409,319.917,-74.080,-176.651,8.310,148.656
C02497=1166.405,320.165,-74.111,-176.648,8.313,148.657
C02498=1166.401,320.413,-74.143,-176.646,8.316,148.657
C02499=1166.397,320.661,-74.175,-176.643,8.319,148.657
C02500=1166.392,320.909,-74.207,-176.641,8.323,148.657
C02501=1166.388,321.157,-74.239,-176.638,8.327,148.657
C02502=1166.385,321.405,-74.271,-176.635,8.330,148.657
C02503=1166.380,321.652,-74.302,-176.633,8.333,148.657
C02504=1166.376,321.901,-74.335,-176.630,8.336,148.657
C02505=1166.372,322.149,-74.366,-176.628,8.339,148.658
C02506=1166.368,322.396,-74.398,-176.626,8.342,148.658
C02507=1166.364,322.644,-74.430,-176.623,8.345,148.658
C02508=1166.360,322.892,-74.462,-176.620,8.349,148.658
C02509=1166.356,323.140,-74.494,-176.618,8.353,148.658
C02510=1166.351,323.388,-74.526,-176.615,8.356,148.658
C02511=1166.347,323.636,-74.558,-176.613,8.359,148.658
C02512=1166.344,323.884,-74.590,-176.611,8.362,148.659
C02513=1166.339,324.132,-74.622,-176.608,8.365,148.659
C02514=1166.335,324.380,-74.654,-176.605,8.369,148.659
C02515=1166.330,324.628,-74.686,-176.603,8.373,148.659
C02516=1166.326,324.876,-74.718,-176.600,8.376,148.659
C02517=1166.323,325.123,-74.750,-176.598,8.379,148.659
C02518=1166.318,325.371,-74.783,-176.595,8.382,148.659
C02519=1166.315,325.619,-74.814,-176.593,8.385,148.659
C02520=1166.310,325.867,-74.847,-176.590,8.389,148.660
C02521=1166.306,326.115,-74.878,-176.588,8.393,148.660
C02522=1166.302,326.363,-74.912,-176.585,8.396,148.660
C02523=1166.298,326.611,-74.943,-176.583,8.399,148.660
C02524=1166.293,326.858,-74.975,-176.580,8.402,148.660
C02525=1166.289,327.106,-75.007,-176.578,8.406,148.661
C02526=1166.285,327.355,-75.040,-176.575,8.408,148.661
C02527=1166.281,327.602,-75.072,-176.572,8.413,148.661
C02528=1166.277,327.851,-75.105,-176.570,8.416,148.661
C02529=1166.273,328.098,-75.136,-176.567,8.419,148.661
C02530=1166.269,328.346,-75.169,-176.565,8.422,148.661
C02531=1166.265,328.594,-75.201,-176.563,8.425,148.661
C02532=1166.260,328.842,-75.234,-176.560,8.429,148.662
C02533=1166.257,329.089,-75.266,-176.557,8.433,148.662
C02534=1166.252,329.337,-75.298,-176.555,8.436,148.662
C02535=1166.248,329.585,-75.330,-176.553,8.439,148.662
C02536=1166.244,329.833,-75.363,-176.550,8.442,148.662
C02537=1166.240,330.081,-75.396,-176.548,8.445,148.662
C02538=1166.236,330.329,-75.428,-176.545,8.449,148.662
C02539=1166.232,330.577,-75.461,-176.542,8.453,148.663
C02540=1166.228,330.824,-75.493,-176.540,8.456,148.663
C02541=1166.223,331.072,-75.525,-176.537,8.459,148.663
C02542=1166.219,331.320,-75.559,-176.535,8.462,148.663
C02543=1166.216,331.568,-75.590,-176.533,8.466,148.663
C02544=1166.211,331.816,-75.624,-176.530,8.470,148.663
C02545=1166.207,332.064,-75.656,-176.528,8.473,148.664
C02546=1166.204,332.311,-75.689,-176.525,8.476,148.664
C02547=1166.199,332.560,-75.721,-176.523,8.479,148.664
C02548=1166.194,332.807,-75.754,-176.520,8.483,148.664
C02549=1166.191,333.055,-75.786,-176.517,8.487,148.664
C02550=1166.187,333.302,-75.819,-176.515,8.490,148.665
C02551=1166.182,333.551,-75.851,-176.512,8.493,148.665
C02552=1166.178,333.799,-75.884,-176.510,8.496,148.665
C02553=1166.175,334.046,-75.917,-176.508,8.500,148.665
C02554=1166.170,334.294,-75.949,-176.505,8.504,148.665
C02555=1166.166,334.542,-75.983,-176.503,8.507,148.665
C02556=1166.162,334.790,-76.016,-176.500,8.510,148.665
C02557=1166.158,335.038,-76.048,-176.498,8.513,148.666
C02558=1166.154,335.286,-76.081,-176.495,8.517,148.666
C02559=1166.150,335.533,-76.114,-176.492,8.521,148.666
C02560=1166.146,335.781,-76.147,-176.490,8.524,148.666
C02561=1166.141,336.029,-76.179,-176.488,8.527,148.666
C02562=1166.138,336.277,-76.212,-176.486,8.531,148.667
C02563=1166.134,336.525,-76.245,-176.482,8.534,148.667
C02564=1166.130,336.772,-76.278,-176.480,8.538,148.667
C02565=1166.125,337.021,-76.311,-176.478,8.541,148.667
C02566=1166.121,337.268,-76.344,-176.475,8.544,148.667
C02567=1166.118,337.516,-76.376,-176.473,8.548,148.668
C02568=1166.113,337.763,-76.410,-176.470,8.552,148.668
C02569=1166.109,338.011,-76.443,-176.468,8.555,148.668
C02570=1166.105,338.259,-76.476,-176.466,8.558,148.668
C02571=1166.101,338.507,-76.508,-176.463,8.561,148.668
C02572=1166.097,338.755,-76.542,-176.460,8.565,148.668
C02573=1166.092,339.003,-76.575,-176.458,8.569,148.669
C02574=1166.088,339.250,-76.608,-176.455,8.572,148.669
C02575=1166.084,339.530,-76.645,-176.453,8.576,148.669
C02576=1166.079,339.809,-76.682,-176.450,8.580,148.669
C02577=1166.075,340.088,-76.719,-176.447,8.583,148.670
C02578=1166.070,340.368,-76.757,-176.445,8.588,148.670
C02579=1166.066,340.616,-76.790,-176.442,8.592,148.670
C02580=1166.062,340.863,-76.823,-176.439,8.595,148.670
C02581=1166.058,341.111,-76.856,-176.437,8.598,148.671
C02582=1166.054,341.359,-76.890,-176.435,8.602,148.671
C02583=1166.050,341.607,-76.923,-176.432,8.605,148.671
C02584=1166.046,341.855,-76.956,-176.429,8.609,148.671
C02585=1166.042,342.103,-76.989,-176.427,8.612,148.671
C02586=1166.038,342.350,-77.023,-176.425,8.615,148.671
C02587=1166.033,342.598,-77.056,-176.422,8.619,148.672
C02588=1166.029,342.846,-77.089,-176.419,8.623,148.672
C02589=1166.025,343.093,-77.123,-176.417,8.626,148.672
C02590=1166.021,343.341,-77.157,-176.415,8.629,148.672
C02591=1166.016,343.589,-77.190,-176.412,8.633,148.673
C02592=1166.012,343.836,-77.223,-176.410,8.637,148.673
C02593=1166.009,344.085,-77.256,-176.407,8.640,148.673
C02594=1166.005,344.333,-77.290,-176.405,8.643,148.673
C02595=1166.001,344.580,-77.323,-176.402,8.647,148.673
C02596=1165.997,344.827,-77.357,-176.400,8.651,148.674
C02597=1165.993,345.075,-77.390,-176.398,8.654,148.674
C02598=1165.988,345.323,-77.423,-176.395,8.658,148.674
C02599=1165.984,345.570,-77.457,-176.393,8.661,148.674
C02600=1165.980,345.819,-77.491,-176.390,8.665,148.675
C02601=1165.976,346.066,-77.524,-176.388,8.668,148.675
C02602=1165.972,346.314,-77.558,-176.385,8.672,148.675
C02603=1165.968,346.561,-77.591,-176.383,8.676,148.675
C02604=1165.964,346.809,-77.624,-176.381,8.679,148.676
C02605=1165.959,347.056,-77.659,-176.378,8.683,148.676
C02606=1165.956,347.305,-77.692,-176.376,8.686,148.676
C02607=1165.952,347.553,-77.725,-176.374,8.690,148.676
C02608=1165.948,347.800,-77.759,-176.371,8.693,148.677
C02609=1165.943,348.048,-77.793,-176.368,8.697,148.677
C02610=1165.939,348.295,-77.827,-176.366,8.700,148.677
C02611=1165.936,348.543,-77.860,-176.364,8.704,148.677
C02612=1165.932,348.791,-77.893,-176.361,8.708,148.678
C02613=1165.927,349.038,-77.928,-176.359,8.711,148.678
C02614=1165.923,349.286,-77.961,-176.356,8.714,148.678
C02615=1165.920,349.534,-77.995,-176.354,8.719,148.678
C02616=1165.915,349.782,-78.029,-176.352,8.722,148.679
C02617=1165.911,350.029,-78.063,-176.349,8.725,148.679
C02618=1165.907,350.276,-78.097,-176.346,8.730,148.679
C02619=1165.904,350.525,-78.130,-176.344,8.733,148.679
C02620=1165.899,350.772,-78.165,-176.342,8.736,148.680
C02621=1165.895,351.020,-78.198,-176.340,8.739,148.680
C02622=1165.892,351.268,-78.232,-176.337,8.743,148.680
C02623=1165.887,351.516,-78.266,-176.335,8.747,148.680
C02624=1165.883,351.763,-78.300,-176.333,8.750,148.681
C02625=1165.879,352.010,-78.334,-176.330,8.755,148.681
C02626=1165.875,352.259,-78.368,-176.327,8.758,148.681
C02627=1165.871,352.506,-78.402,-176.325,8.761,148.681
C02628=1165.867,352.753,-78.436,-176.323,8.766,148.682
C02629=1165.863,353.002,-78.470,-176.320,8.769,148.682
C02630=1165.859,353.249,-78.504,-176.318,8.772,148.682
C02631=1165.854,353.496,-78.538,-176.315,8.776,148.682
C02632=1165.851,353.744,-78.572,-176.313,8.780,148.683
C02633=1165.846,353.992,-78.606,-176.310,8.784,148.683
C02634=1165.843,354.239,-78.640,-176.308,8.787,148.683
C02635=1165.839,354.487,-78.674,-176.306,8.791,148.684
C02636=1165.835,354.734,-78.709,-176.303,8.795,148.684
C02637=1165.831,354.981,-78.742,-176.301,8.798,148.684
C02638=1165.827,355.230,-78.777,-176.299,8.802,148.685
C02639=1165.823,355.477,-78.810,-176.296,8.806,148.685
C02640=1165.819,355.725,-78.845,-176.294,8.809,148.685
C02641=1165.815,355.972,-78.879,-176.291,8.812,148.685
C02642=1165.810,356.220,-78.914,-176.289,8.817,148.686
C02643=1165.807,356.468,-78.948,-176.287,8.820,148.686
C02644=1165.803,356.715,-78.982,-176.284,8.823,148.686
C02645=1165.799,356.964,-79.016,-176.282,8.828,148.687
C02646=1165.794,357.211,-79.050,-176.280,8.831,148.687
C02647=1165.791,357.458,-79.084,-176.277,8.835,148.687
C02648=1165.787,357.706,-79.119,-176.275,8.839,148.688
C02649=1165.782,357.954,-79.153,-176.273,8.842,148.688
C02650=1165.779,358.201,-79.188,-176.270,8.846,148.688
C02651=1165.774,358.449,-79.222,-176.267,8.849,148.688
C02652=1165.771,358.697,-79.256,-176.265,8.854,148.689
C02653=1165.767,358.944,-79.291,-176.263,8.857,148.689
C02654=1165.763,359.191,-79.325,-176.261,8.861,148.689
C02655=1165.759,359.439,-79.360,-176.258,8.865,148.690
C02656=1165.754,359.686,-79.395,-176.256,8.868,148.690
C02657=1165.751,359.934,-79.429,-176.253,8.873,148.690
C02658=1165.747,360.181,-79.463,-176.251,8.876,148.691
C02659=1165.743,360.429,-79.498,-176.249,8.879,148.691
C02660=1165.739,360.677,-79.532,-176.246,8.884,148.691
C02661=1165.735,360.925,-79.567,-176.244,8.887,148.691
C02662=1165.730,361.172,-79.601,-176.242,8.891,148.692
C02663=1165.727,361.419,-79.636,-176.239,8.895,148.692
C02664=1165.723,361.667,-79.671,-176.237,8.898,148.693
C02665=1165.719,361.915,-79.706,-176.235,8.902,148.693
C02666=1165.715,362.162,-79.740,-176.233,8.906,148.693
C02667=1165.711,362.410,-79.774,-176.230,8.910,148.694
C02668=1165.707,362.657,-79.810,-176.228,8.914,148.694
C02669=1165.703,362.905,-79.844,-176.226,8.917,148.694
C02670=1165.700,363.153,-79.879,-176.223,8.921,148.695
C02671=1165.695,363.400,-79.913,-176.221,8.925,148.695
C02672=1165.691,363.648,-79.949,-176.219,8.929,148.695
C02673=1165.687,363.895,-79.983,-176.216,8.932,148.696
C02674=1165.684,364.143,-80.017,-176.214,8.936,148.696
C02675=1165.679,364.390,-80.053,-176.212,8.940,148.696
C02676=1165.675,364.638,-80.087,-176.210,8.944,148.697
C02677=1165.672,364.885,-80.123,-176.208,8.947,148.697
C02678=1165.668,365.132,-80.157,-176.205,8.952,148.698
C02679=1165.663,365.415,-80.197,-176.202,8.956,148.698
C02680=1165.659,365.697,-80.237,-176.200,8.960,148.698
C02681=1165.654,365.980,-80.277,-176.198,8.965,148.699
C02682=1165.650,366.262,-80.317,-176.195,8.969,148.699
C02683=1165.645,366.510,-80.351,-176.193,8.973,148.700
C02684=1165.641,366.758,-80.386,-176.191,8.976,148.700
C02685=1165.637,367.005,-80.421,-176.189,8.981,148.701
C02686=1165.633,367.253,-80.456,-176.187,8.984,148.701
C02687=1165.630,367.500,-80.492,-176.185,8.988,148.701
C02688=1165.626,367.747,-80.526,-176.182,8.992,148.702
C02689=1165.622,367.995,-80.561,-176.181,8.996,148.702
C02690=1165.618,368.242,-80.597,-176.179,8.999,148.703
C02691=1165.614,368.490,-80.631,-176.177,9.003,148.703
C02692=1165.610,368.737,-80.667,-176.174,9.007,148.703
C02693=1165.606,368.985,-80.701,-176.173,9.011,148.704
C02694=1165.602,369.232,-80.737,-176.171,9.014,148.704
C02695=1165.598,369.480,-80.772,-176.168,9.019,148.705
C02696=1165.594,369.728,-80.807,-176.166,9.022,148.705
C02697=1165.590,369.975,-80.842,-176.165,9.026,148.706
C02698=1165.586,370.222,-80.878,-176.163,9.030,148.706
C02699=1165.582,370.470,-80.913,-176.161,9.034,148.707
C02700=1165.578,370.717,-80.948,-176.159,9.038,148.707
C02701=1165.574,370.964,-80.983,-176.157,9.042,148.708
C02702=1165.570,371.213,-81.018,-176.156,9.045,148.708
C02703=1165.566,371.459,-81.053,-176.154,9.049,148.709
C02704=1165.563,371.707,-81.089,-176.152,9.053,148.709
C02705=1165.559,371.954,-81.124,-176.150,9.057,148.710
C02706=1165.555,372.202,-81.159,-176.149,9.060,148.710
C02707=1165.551,372.449,-81.194,-176.146,9.065,148.711
C02708=1165.547,372.697,-81.230,-176.145,9.069,148.711
C02709=1165.543,372.944,-81.265,-176.143,9.072,148.712
C02710=1165.539,373.192,-81.300,-176.141,9.076,148.712
C02711=1165.534,373.439,-81.336,-176.140,9.080,148.713
C02712=1165.531,373.687,-81.372,-176.138,9.084,148.713
C02713=1165.527,373.935,-81.407,-176.136,9.087,148.714
C02714=1165.523,374.181,-81.442,-176.135,9.091,148.714
C02715=1165.519,374.429,-81.478,-176.133,9.095,148.715
C02716=1165.515,374.676,-81.513,-176.131,9.099,148.715
C02717=1165.511,374.924,-81.548,-176.130,9.102,148.716
C02718=1165.508,375.172,-81.584,-176.129,9.106,148.717
C02719=1165.504,375.419,-81.619,-176.127,9.110,148.717
C02720=1165.499,375.667,-81.655,-176.126,9.113,148.718
C02721=1165.496,375.914,-81.691,-176.124,9.117,148.718
C02722=1165.492,376.162,-81.726,-176.123,9.121,148.719
C02723=1165.488,376.408,-81.761,-176.122,9.125,148.720
C02724=1165.484,376.656,-81.797,-176.120,9.129,148.720
C02725=1165.480,376.903,-81.833,-176.119,9.133,148.721
C02726=1165.476,377.151,-81.869,-176.117,9.136,148.721
C02727=1165.472,377.399,-81.904,-176.116,9.140,148.722
C02728=1165.468,377.645,-81.939,-176.115,9.143,148.723
C02729=1165.464,377.893,-81.975,-176.114,9.147,148.723
C02730=1165.461,378.140,-82.010,-176.112,9.151,148.724
C02731=1165.456,378.388,-82.047,-176.111,9.154,148.725
C02732=1165.453,378.636,-82.082,-176.110,9.158,148.725
C02733=1165.449,378.883,-82.118,-176.108,9.162,148.726
C02734=1165.445,379.130,-82.153,-176.108,9.165,148.726
C02735=1165.440,379.378,-82.189,-176.107,9.169,148.727
C02736=1165.437,379.625,-82.225,-176.106,9.173,148.728
C02737=1165.433,379.872,-82.261,-176.104,9.176,148.728
C02738=1165.429,380.120,-82.297,-176.104,9.180,148.729
C02739=1165.425,380.368,-82.333,-176.102,9.184,148.730
C02740=1165.421,380.614,-82.368,-176.102,9.187,148.730
C02741=1165.417,380.862,-82.403,-176.101,9.191,148.731
C02742=1165.413,381.110,-82.439,-176.100,9.194,148.732
C02743=1165.409,381.357,-82.476,-176.099,9.198,148.733
C02744=1165.406,381.604,-82.511,-176.098,9.201,148.733
C02745=1165.401,381.852,-82.547,-176.097,9.206,148.734
C02746=1165.398,382.099,-82.583,-176.096,9.209,148.735
C02747=1165.394,382.347,-82.618,-176.096,9.212,148.735
C02748=1165.389,382.594,-82.654,-176.094,9.216,148.736
C02749=1165.386,382.841,-82.691,-176.094,9.219,148.737
C02750=1165.382,383.088,-82.726,-176.093,9.223,148.737
C02751=1165.378,383.336,-82.762,-176.092,9.226,148.738
C02752=1165.374,383.584,-82.798,-176.092,9.229,148.739
C02753=1165.371,383.831,-82.834,-176.091,9.233,148.740
C02754=1165.366,384.078,-82.870,-176.091,9.237,148.740
C02755=1165.363,384.326,-82.906,-176.090,9.240,148.741
C02756=1165.359,384.573,-82.942,-176.089,9.243,148.742
C02757=1165.354,384.820,-82.978,-176.089,9.247,148.742
C02758=1165.351,385.067,-83.013,-176.088,9.250,148.743
C02759=1165.347,385.315,-83.049,-176.088,9.254,148.744
C02760=1165.343,385.562,-83.086,-176.088,9.257,148.745
C02761=1165.339,385.810,-83.121,-176.087,9.260,148.746
C02762=1165.335,386.057,-83.157,-176.087,9.264,148.746
C02763=1165.331,386.304,-83.194,-176.086,9.267,148.747
C02764=1165.328,386.552,-83.229,-176.086,9.270,148.748
C02765=1165.323,386.800,-83.265,-176.086,9.273,148.749
C02766=1165.320,387.046,-83.302,-176.086,9.276,148.749
C02767=1165.316,387.294,-83.338,-176.085,9.280,148.750
C02768=1165.312,387.542,-83.373,-176.085,9.282,148.751
C02769=1165.309,387.789,-83.410,-176.085,9.286,148.752
C02770=1165.304,388.036,-83.446,-176.084,9.289,148.752
C02771=1165.301,388.283,-83.482,-176.085,9.292,148.753
C02772=1165.296,388.530,-83.518,-176.084,9.295,148.754
C02773=1165.292,388.778,-83.553,-176.084,9.298,148.755
C02774=1165.288,389.025,-83.590,-176.084,9.301,148.755
C02775=1165.284,389.273,-83.626,-176.084,9.304,148.756
C02776=1165.280,389.520,-83.663,-176.084,9.307,148.757
C02777=1165.277,389.767,-83.698,-176.084,9.310,148.758
C02778=1165.273,390.015,-83.734,-176.084,9.312,148.758
C02779=1165.269,390.262,-83.771,-176.084,9.316,148.759
C02780=1165.265,390.509,-83.806,-176.084,9.319,148.760
C02781=1165.261,390.757,-83.843,-176.085,9.321,148.761
C02782=1165.257,391.004,-83.878,-176.084,9.325,148.762
C02783=1165.253,391.289,-83.921,-176.085,9.328,148.763
C02784=1165.248,391.575,-83.962,-176.085,9.331,148.763
C02785=1165.244,391.860,-84.004,-176.085,9.334,148.764
C02786=1165.240,392.145,-84.046,-176.085,9.338,148.765
C02787=1165.236,392.392,-84.082,-176.085,9.340,148.766
C02788=1165.232,392.640,-84.118,-176.086,9.343,148.767
C02789=1165.228,392.887,-84.154,-176.086,9.346,148.767
C02790=1165.224,393.135,-84.191,-176.086,9.348,148.768
C02791=1165.220,393.382,-84.226,-176.086,9.351,148.769
C02792=1165.216,393.630,-84.263,-176.087,9.354,148.770
C02793=1165.213,393.877,-84.298,-176.087,9.356,148.771
C02794=1165.209,394.124,-84.335,-176.087,9.359,148.771
C02795=1165.205,394.372,-84.371,-176.087,9.362,148.772
C02796=1165.201,394.619,-84.408,-176.088,9.364,148.773
C02797=1165.197,394.866,-84.444,-176.088,9.367,148.774
C02798=1165.193,395.114,-84.480,-176.088,9.370,148.774
C02799=1165.190,395.361,-84.516,-176.088,9.372,148.775
C02800=1165.185,395.608,-84.553,-176.089,9.375,148.776
C02801=1165.182,395.855,-84.589,-176.089,9.376,148.777
C02802=1165.178,396.103,-84.625,-176.090,9.379,148.777
C02803=1165.173,396.350,-84.662,-176.090,9.382,148.778
C02804=1165.170,396.598,-84.697,-176.090,9.384,148.779
C02805=1165.165,396.844,-84.734,-176.091,9.387,148.780
C02806=1165.161,397.092,-84.769,-176.091,9.389,148.780
C02807=1165.157,397.339,-84.806,-176.091,9.392,148.781
C02808=1165.154,397.586,-84.842,-176.092,9.394,148.782
C02809=1165.150,397.834,-84.879,-176.092,9.396,148.783
C02810=1165.147,398.081,-84.915,-176.093,9.399,148.783
C02811=1165.142,398.329,-84.951,-176.093,9.401,148.784
C02812=1165.139,398.576,-84.988,-176.094,9.403,148.785
C02813=1165.135,398.824,-85.024,-176.094,9.406,148.785
C02814=1165.131,399.071,-85.060,-176.095,9.408,148.786
C02815=1165.127,399.318,-85.096,-176.095,9.410,148.787
C02816=1165.123,399.566,-85.133,-176.095,9.413,148.788
C02817=1165.119,399.813,-85.169,-176.096,9.415,148.788
C02818=1165.115,400.060,-85.206,-176.096,9.417,148.789
C02819=1165.112,400.307,-85.242,-176.097,9.419,148.790
C02820=1165.107,400.555,-85.278,-176.097,9.422,148.791
C02821=1165.104,400.802,-85.314,-176.098,9.424,148.791
C02822=1165.100,401.050,-85.350,-176.098,9.426,148.792
C02823=1165.096,401.296,-85.387,-176.099,9.428,148.793
C02824=1165.092,401.544,-85.423,-176.099,9.430,148.793
C02825=1165.088,401.791,-85.460,-176.100,9.432,148.794
C02826=1165.084,402.038,-85.496,-176.101,9.434,148.795
C02827=1165.080,402.286,-85.532,-176.101,9.437,148.795
C02828=1165.077,402.533,-85.568,-176.101,9.438,148.796
C02829=1165.072,402.780,-85.605,-176.102,9.441,148.797
C02830=1165.069,403.028,-85.641,-176.102,9.443,148.797
C02831=1165.065,403.275,-85.678,-176.103,9.445,148.798
C02832=1165.060,403.523,-85.714,-176.103,9.447,148.799
C02833=1165.057,403.770,-85.750,-176.104,9.449,148.800
C02834=1165.053,404.017,-85.787,-176.104,9.452,148.800
C02835=1165.049,404.264,-85.822,-176.105,9.453,148.801
C02836=1165.045,404.512,-85.859,-176.106,9.455,148.802
C02837=1165.042,404.758,-85.895,-176.106,9.458,148.802
C02838=1165.037,405.006,-85.932,-176.106,9.459,148.803
C02839=1165.033,405.253,-85.968,-176.107,9.461,148.803
C02840=1165.030,405.501,-86.004,-176.107,9.463,148.804
C02841=1165.026,405.748,-86.041,-176.108,9.465,148.805
C02842=1165.022,405.995,-86.077,-176.108,9.467,148.805
C02843=1165.018,406.243,-86.113,-176.109,9.469,148.806
C02844=1165.014,406.490,-86.150,-176.109,9.471,148.807
C02845=1165.010,406.737,-86.186,-176.110,9.473,148.807
C02846=1165.006,406.985,-86.223,-176.111,9.475,148.808
C02847=1165.003,407.232,-86.259,-176.111,9.477,148.809
C02848=1164.998,407.479,-86.296,-176.111,9.479,148.809
C02849=1164.994,407.727,-86.332,-176.112,9.480,148.810
C02850=1164.991,407.973,-86.368,-176.112,9.482,148.811
C02851=1164.987,408.221,-86.405,-176.113,9.485,148.811
C02852=1164.984,408.469,-86.441,-176.113,9.486,148.812
C02853=1164.979,408.716,-86.478,-176.114,9.488,148.813
C02854=1164.976,408.964,-86.513,-176.114,9.490,148.813
C02855=1164.972,409.211,-86.550,-176.115,9.491,148.814
C02856=1164.968,409.458,-86.587,-176.115,9.494,148.814
C02857=1164.964,409.705,-86.623,-176.116,9.496,148.815
C02858=1164.960,409.953,-86.659,-176.116,9.497,148.816
C02859=1164.956,410.200,-86.696,-176.117,9.499,148.816
C02860=1164.952,410.447,-86.732,-176.117,9.501,148.817
C02861=1164.948,410.694,-86.769,-176.118,9.503,148.818
C02862=1164.945,410.941,-86.805,-176.118,9.505,148.818
C02863=1164.941,411.189,-86.842,-176.119,9.506,148.819
C02864=1164.936,411.436,-86.878,-176.119,9.508,148.819
C02865=1164.933,411.683,-86.914,-176.119,9.510,148.820
C02866=1164.929,411.930,-86.951,-176.120,9.512,148.820
C02867=1164.925,412.178,-86.987,-176.120,9.514,148.821
C02868=1164.921,412.425,-87.023,-176.121,9.515,148.822
C02869=1164.917,412.672,-87.060,-176.121,9.517,148.822
C02870=1164.913,412.920,-87.096,-176.122,9.520,148.823
C02871=1164.909,413.167,-87.133,-176.122,9.521,148.823
C02872=1164.905,413.414,-87.170,-176.123,9.523,148.824
C02873=1164.901,413.662,-87.205,-176.123,9.524,148.824
C02874=1164.898,413.910,-87.242,-176.124,9.526,148.825
C02875=1164.894,414.156,-87.279,-176.123,9.528,148.826
C02876=1164.890,414.404,-87.315,-176.124,9.530,148.826
C02877=1164.886,414.651,-87.352,-176.125,9.532,148.827
C02878=1164.883,414.898,-87.388,-176.125,9.533,148.827
C02879=1164.879,415.146,-87.425,-176.126,9.535,148.828
C02880=1164.875,415.393,-87.460,-176.125,9.537,148.828
C02881=1164.872,415.641,-87.497,-176.126,9.539,148.829
C02882=1164.870,415.887,-87.534,-176.126,9.540,148.830
C02883=1164.870,416.215,-87.581,-176.127,9.542,148.830
C02884=1164.871,416.540,-87.628,-176.127,9.545,148.831
C02885=1164.873,416.867,-87.676,-176.128,9.546,148.832
C02886=1164.877,417.193,-87.723,-176.128,9.549,148.832
C02887=1164.456,417.195,-87.769,-176.131,9.560,148.836
C02888=1164.453,416.865,-87.721,-176.130,9.558,148.835
C02889=1164.450,416.536,-87.673,-176.130,9.556,148.835
C02890=1164.449,416.206,-87.626,-176.130,9.554,148.834
C02891=1164.450,415.876,-87.577,-176.129,9.551,148.833
C02892=1164.451,415.629,-87.541,-176.129,9.550,148.833
C02893=1164.454,415.382,-87.504,-176.129,9.548,148.832
C02894=1164.457,415.134,-87.469,-176.128,9.546,148.832
C02895=1164.462,414.887,-87.432,-176.128,9.544,148.831
C02896=1164.466,414.640,-87.395,-176.127,9.542,148.830
C02897=1164.468,414.392,-87.358,-176.127,9.541,148.830
C02898=1164.473,414.145,-87.322,-176.126,9.539,148.829
C02899=1164.477,413.897,-87.285,-176.126,9.537,148.829
C02900=1164.480,413.651,-87.249,-176.126,9.535,148.828
C02901=1164.485,413.403,-87.213,-176.125,9.533,148.828
C02902=1164.488,413.156,-87.177,-176.125,9.532,148.827
C02903=1164.492,412.909,-87.140,-176.124,9.530,148.826
C02904=1164.497,412.661,-87.104,-176.124,9.529,148.826
C02905=1164.500,412.414,-87.068,-176.124,9.526,148.825
C02906=1164.504,412.167,-87.031,-176.123,9.525,148.825
C02907=1164.508,411.920,-86.994,-176.123,9.523,148.824
C02908=1164.512,411.672,-86.958,-176.122,9.521,148.824
C02909=1164.516,411.425,-86.921,-176.122,9.520,148.823
C02910=1164.519,411.178,-86.885,-176.121,9.517,148.822
C02911=1164.524,410.930,-86.849,-176.121,9.516,148.822
C02912=1164.528,410.683,-86.812,-176.120,9.514,148.821
C02913=1164.531,410.436,-86.776,-176.120,9.512,148.820
C02914=1164.535,410.188,-86.740,-176.119,9.510,148.820
C02915=1164.540,409.941,-86.703,-176.119,9.508,148.819
C02916=1164.542,409.694,-86.666,-176.119,9.506,148.819
C02917=1164.547,409.446,-86.630,-176.118,9.505,148.818
C02918=1164.550,409.199,-86.594,-176.117,9.503,148.817
C02919=1164.554,408.952,-86.557,-176.117,9.501,148.817
C02920=1164.559,408.704,-86.521,-176.117,9.499,148.816
C02921=1164.562,408.457,-86.485,-176.116,9.497,148.816
C02922=1164.566,408.210,-86.448,-176.115,9.495,148.815
C02923=1164.570,407.962,-86.412,-176.115,9.494,148.814
C02924=1164.574,407.715,-86.375,-176.115,9.491,148.813
C02925=1164.578,407.468,-86.338,-176.114,9.490,148.813
C02926=1164.581,407.220,-86.303,-176.114,9.488,148.812
C02927=1164.586,406.973,-86.266,-176.113,9.486,148.812
C02928=1164.589,406.726,-86.230,-176.113,9.484,148.811
C02929=1164.593,406.479,-86.194,-176.112,9.482,148.810
C02930=1164.597,406.231,-86.157,-176.111,9.480,148.810
C02931=1164.601,405.984,-86.121,-176.111,9.478,148.809
C02932=1164.605,405.737,-86.084,-176.111,9.476,148.808
C02933=1164.609,405.490,-86.048,-176.110,9.474,148.808
C02934=1164.613,405.243,-86.011,-176.109,9.472,148.807
C02935=1164.617,404.995,-85.975,-176.109,9.470,148.806
C02936=1164.620,404.748,-85.939,-176.108,9.468,148.806
C02937=1164.624,404.501,-85.902,-176.108,9.466,148.805
C02938=1164.628,404.253,-85.866,-176.107,9.464,148.804
C02939=1164.632,404.006,-85.830,-176.107,9.462,148.804
C02940=1164.635,403.758,-85.794,-176.106,9.460,148.803
C02941=1164.639,403.511,-85.757,-176.106,9.458,148.802
C02942=1164.643,403.263,-85.720,-176.105,9.456,148.802
C02943=1164.647,403.016,-85.684,-176.104,9.454,148.801
C02944=1164.651,402.769,-85.648,-176.104,9.452,148.800
C02945=1164.655,402.522,-85.611,-176.104,9.450,148.800
C02946=1164.659,402.274,-85.575,-176.103,9.447,148.799
C02947=1164.662,402.027,-85.539,-176.103,9.445,148.798
C02948=1164.667,401.779,-85.503,-176.102,9.444,148.798
C02949=1164.671,401.532,-85.466,-176.102,9.441,148.797
C02950=1164.674,401.285,-85.430,-176.101,9.439,148.796
C02951=1164.679,401.037,-85.393,-176.101,9.437,148.795
C02952=1164.682,400.791,-85.357,-176.100,9.435,148.795
C02953=1164.686,400.543,-85.321,-176.100,9.432,148.794
C02954=1164.690,400.296,-85.285,-176.099,9.430,148.793
C02955=1164.694,400.049,-85.248,-176.099,9.428,148.793
C02956=1164.698,399.801,-85.212,-176.098,9.426,148.792
C02957=1164.702,399.554,-85.176,-176.098,9.423,148.791
C02958=1164.706,399.306,-85.139,-176.097,9.422,148.790
C02959=1164.709,399.059,-85.103,-176.097,9.419,148.790
C02960=1164.713,398.812,-85.066,-176.096,9.417,148.789
C02961=1164.717,398.565,-85.031,-176.096,9.415,148.788
C02962=1164.721,398.317,-84.994,-176.095,9.412,148.788
C02963=1164.725,398.070,-84.958,-176.095,9.410,148.787
C02964=1164.729,397.823,-84.921,-176.095,9.407,148.786
C02965=1164.733,397.575,-84.885,-176.094,9.405,148.785
C02966=1164.737,397.328,-84.849,-176.093,9.403,148.785
C02967=1164.741,397.081,-84.812,-176.093,9.400,148.784
C02968=1164.744,396.833,-84.777,-176.093,9.398,148.783
C02969=1164.749,396.586,-84.740,-176.092,9.396,148.783
C02970=1164.752,396.339,-84.704,-176.092,9.393,148.782
C02971=1164.756,396.092,-84.667,-176.092,9.391,148.781
C02972=1164.760,395.844,-84.632,-176.092,9.388,148.780
C02973=1164.764,395.597,-84.595,-176.090,9.386,148.779
C02974=1164.768,395.349,-84.559,-176.090,9.383,148.779
C02975=1164.772,395.102,-84.523,-176.090,9.381,148.778
C02976=1164.776,394.854,-84.486,-176.090,9.378,148.777
C02977=1164.780,394.607,-84.450,-176.089,9.375,148.776
C02978=1164.784,394.360,-84.413,-176.089,9.373,148.776
C02979=1164.787,394.113,-84.378,-176.089,9.370,148.775
C02980=1164.791,393.866,-84.341,-176.089,9.367,148.774
C02981=1164.795,393.618,-84.305,-176.088,9.365,148.773
C02982=1164.799,393.371,-84.269,-176.088,9.362,148.773
C02983=1164.803,393.123,-84.233,-176.088,9.359,148.772
C02984=1164.807,392.876,-84.196,-176.088,9.357,148.771
C02985=1164.811,392.629,-84.161,-176.087,9.354,148.770
C02986=1164.815,392.381,-84.124,-176.087,9.351,148.769
C02987=1164.818,392.134,-84.088,-176.087,9.349,148.769
C02988=1164.822,391.849,-84.046,-176.086,9.346,148.768
C02989=1164.827,391.564,-84.005,-176.087,9.342,148.767
C02990=1164.832,391.278,-83.963,-176.087,9.339,148.766
C02991=1164.836,390.993,-83.921,-176.086,9.336,148.765
C02992=1164.840,390.745,-83.885,-176.086,9.333,148.764
C02993=1164.844,390.498,-83.849,-176.086,9.330,148.764
C02994=1164.848,390.250,-83.813,-176.086,9.327,148.763
C02995=1164.852,390.003,-83.776,-176.086,9.324,148.762
C02996=1164.855,389.756,-83.741,-176.086,9.321,148.761
C02997=1164.860,389.509,-83.704,-176.086,9.319,148.760
C02998=1164.864,389.262,-83.669,-176.086,9.315,148.760
C02999=1164.868,389.014,-83.632,-176.086,9.312,148.759
C03000=1164.871,388.767,-83.596,-176.086,9.310,148.758
C03001=1164.875,388.520,-83.561,-176.086,9.306,148.757
C03002=1164.879,388.272,-83.524,-176.086,9.303,148.757
C03003=1164.883,388.025,-83.488,-176.086,9.300,148.756
C03004=1164.887,387.778,-83.451,-176.086,9.297,148.755
C03005=1164.891,387.530,-83.416,-176.086,9.294,148.754
C03006=1164.895,387.282,-83.380,-176.087,9.291,148.753
C03007=1164.898,387.036,-83.343,-176.087,9.287,148.753
C03008=1164.902,386.788,-83.308,-176.087,9.284,148.752
C03009=1164.906,386.540,-83.272,-176.087,9.281,148.751
C03010=1164.910,386.293,-83.235,-176.088,9.278,148.750
C03011=1164.914,386.046,-83.199,-176.088,9.275,148.750
C03012=1164.918,385.798,-83.164,-176.089,9.271,148.749
C03013=1164.921,385.551,-83.127,-176.089,9.268,148.748
C03014=1164.926,385.303,-83.091,-176.089,9.264,148.747
C03015=1164.930,385.057,-83.056,-176.090,9.261,148.747
C03016=1164.934,384.809,-83.019,-176.090,9.258,148.746
C03017=1164.938,384.562,-82.984,-176.091,9.255,148.745
C03018=1164.941,384.314,-82.948,-176.092,9.251,148.744
C03019=1164.945,384.067,-82.911,-176.092,9.248,148.744
C03020=1164.949,383.820,-82.876,-176.092,9.244,148.743
C03021=1164.953,383.572,-82.840,-176.093,9.241,148.742
C03022=1164.957,383.324,-82.804,-176.094,9.238,148.742
C03023=1164.960,383.077,-82.768,-176.095,9.234,148.741
C03024=1164.965,382.830,-82.732,-176.095,9.230,148.740
C03025=1164.969,382.582,-82.696,-176.096,9.227,148.739
C03026=1164.973,382.335,-82.661,-176.097,9.223,148.739
C03027=1164.977,382.088,-82.624,-176.098,9.220,148.738
C03028=1164.981,381.841,-82.589,-176.098,9.217,148.737
C03029=1164.984,381.593,-82.553,-176.099,9.212,148.736
C03030=1164.988,381.346,-82.517,-176.100,9.209,148.736
C03031=1164.992,381.098,-82.481,-176.101,9.206,148.735
C03032=1164.996,380.851,-82.445,-176.102,9.202,148.734
C03033=1164.999,380.603,-82.409,-176.103,9.199,148.734
C03034=1165.004,380.356,-82.374,-176.104,9.195,148.733
C03035=1165.008,380.109,-82.338,-176.105,9.192,148.732
C03036=1165.012,379.861,-82.303,-176.106,9.187,148.732
C03037=1165.016,379.614,-82.266,-176.107,9.183,148.731
C03038=1165.020,379.366,-82.231,-176.108,9.180,148.730
C03039=1165.023,379.119,-82.195,-176.110,9.176,148.730
C03040=1165.027,378.872,-82.159,-176.110,9.173,148.729
C03041=1165.032,378.625,-82.123,-176.111,9.169,148.728
C03042=1165.035,378.377,-82.088,-176.113,9.165,148.728
C03043=1165.039,378.130,-82.052,-176.114,9.162,148.727
C03044=1165.043,377.882,-82.017,-176.115,9.158,148.727
C03045=1165.047,377.634,-81.981,-176.117,9.154,148.726
C03046=1165.051,377.387,-81.945,-176.118,9.150,148.725
C03047=1165.055,377.140,-81.910,-176.119,9.147,148.725
C03048=1165.059,376.892,-81.874,-176.120,9.143,148.724
C03049=1165.062,376.645,-81.839,-176.122,9.140,148.723
C03050=1165.067,376.397,-81.803,-176.123,9.136,148.723
C03051=1165.071,376.150,-81.767,-176.125,9.132,148.722
C03052=1165.075,375.903,-81.732,-176.126,9.128,148.722
C03053=1165.078,375.655,-81.696,-176.127,9.124,148.721
C03054=1165.082,375.408,-81.661,-176.129,9.120,148.721
C03055=1165.086,375.160,-81.625,-176.131,9.116,148.720
C03056=1165.091,374.913,-81.589,-176.132,9.113,148.719
C03057=1165.094,374.666,-81.554,-176.133,9.110,148.719
C03058=1165.098,374.418,-81.518,-176.135,9.106,148.718
C03059=1165.102,374.170,-81.483,-176.136,9.102,148.718
C03060=1165.106,373.923,-81.448,-176.138,9.098,148.717
C03061=1165.110,373.676,-81.413,-176.140,9.094,148.717
C03062=1165.114,373.428,-81.377,-176.141,9.091,148.716
C03063=1165.117,373.181,-81.342,-176.143,9.086,148.716
C03064=1165.121,372.934,-81.306,-176.145,9.083,148.715
C03065=1165.125,372.686,-81.272,-176.147,9.079,148.714
C03066=1165.130,372.438,-81.236,-176.149,9.075,148.714
C03067=1165.134,372.191,-81.200,-176.150,9.071,148.713
C03068=1165.138,371.944,-81.165,-176.152,9.068,148.713
C03069=1165.141,371.696,-81.129,-176.154,9.064,148.713
C03070=1165.145,371.448,-81.094,-176.155,9.060,148.712
C03071=1165.149,371.201,-81.059,-176.158,9.056,148.711
C03072=1165.153,370.954,-81.024,-176.159,9.052,148.711
C03073=1165.157,370.706,-80.988,-176.161,9.048,148.710
C03074=1165.161,370.458,-80.953,-176.163,9.044,148.710
C03075=1165.165,370.211,-80.918,-176.165,9.041,148.710
C03076=1165.169,369.964,-80.883,-176.167,9.036,148.709
C03077=1165.173,369.716,-80.848,-176.169,9.033,148.709
C03078=1165.177,369.469,-80.813,-176.171,9.029,148.708
C03079=1165.181,369.222,-80.777,-176.173,9.026,148.708
C03080=1165.185,368.973,-80.742,-176.175,9.021,148.707
C03081=1165.189,368.727,-80.707,-176.177,9.018,148.707
C03082=1165.193,368.478,-80.672,-176.179,9.014,148.706
C03083=1165.197,368.231,-80.637,-176.181,9.010,148.706
C03084=1165.201,367.984,-80.601,-176.183,9.006,148.706
C03085=1165.204,367.736,-80.567,-176.185,9.002,148.705
C03086=1165.208,367.489,-80.532,-176.187,8.999,148.705
C03087=1165.212,367.241,-80.497,-176.189,8.994,148.704
C03088=1165.216,366.994,-80.462,-176.191,8.991,148.704
C03089=1165.221,366.747,-80.427,-176.193,8.987,148.703
C03090=1165.224,366.499,-80.392,-176.195,8.983,148.703
C03091=1165.228,366.251,-80.357,-176.198,8.979,148.703
C03092=1165.233,365.969,-80.317,-176.200,8.975,148.702
C03093=1165.237,365.686,-80.277,-176.203,8.971,148.702
C03094=1165.242,365.405,-80.238,-176.205,8.966,148.701
C03095=1165.247,365.122,-80.197,-176.207,8.962,148.701
C03096=1165.250,364.874,-80.163,-176.210,8.958,148.701
C03097=1165.254,364.627,-80.128,-176.212,8.954,148.700
C03098=1165.258,364.379,-80.093,-176.214,8.950,148.700
C03099=1165.262,364.131,-80.058,-176.216,8.947,148.699
C03100=1165.266,363.885,-80.024,-176.219,8.943,148.699
C03101=1165.270,363.636,-79.989,-176.221,8.939,148.699
C03102=1165.274,363.389,-79.954,-176.224,8.935,148.698
C03103=1165.278,363.142,-79.919,-176.225,8.931,148.698
C03104=1165.282,362.894,-79.884,-176.228,8.928,148.698
C03105=1165.286,362.646,-79.850,-176.230,8.924,148.697
C03106=1165.290,362.398,-79.815,-176.232,8.920,148.697
C03107=1165.294,362.151,-79.780,-176.235,8.916,148.696
C03108=1165.297,361.904,-79.746,-176.237,8.913,148.696
C03109=1165.302,361.656,-79.711,-176.240,8.908,148.696
C03110=1165.306,361.408,-79.677,-176.242,8.905,148.696
C03111=1165.310,361.161,-79.641,-176.244,8.901,148.695
C03112=1165.313,360.913,-79.607,-176.247,8.897,148.695
C03113=1165.318,360.666,-79.573,-176.249,8.894,148.695
C03114=1165.322,360.418,-79.538,-176.251,8.890,148.694
C03115=1165.326,360.171,-79.504,-176.254,8.886,148.694
C03116=1165.330,359.923,-79.469,-176.255,8.883,148.694
C03117=1165.333,359.676,-79.435,-176.258,8.879,148.693
C03118=1165.337,359.427,-79.400,-176.261,8.875,148.693
C03119=1165.342,359.181,-79.365,-176.263,8.871,148.693
C03120=1165.345,358.933,-79.331,-176.265,8.868,148.692
C03121=1165.349,358.685,-79.296,-176.268,8.864,148.692
C03122=1165.354,358.438,-79.262,-176.270,8.860,148.692
C03123=1165.357,358.190,-79.228,-176.272,8.857,148.691
C03124=1165.362,357.943,-79.193,-176.275,8.852,148.691
C03125=1165.365,357.695,-79.159,-176.277,8.849,148.691
C03126=1165.370,357.447,-79.125,-176.279,8.846,148.691
C03127=1165.373,357.200,-79.090,-176.282,8.841,148.690
C03128=1165.377,356.952,-79.056,-176.284,8.838,148.690
C03129=1165.381,356.705,-79.023,-176.287,8.834,148.690
C03130=1165.385,356.456,-78.988,-176.289,8.830,148.689
C03131=1165.389,356.209,-78.954,-176.292,8.827,148.689
C03132=1165.393,355.961,-78.919,-176.294,8.823,148.689
C03133=1165.397,355.714,-78.885,-176.296,8.819,148.688
C03134=1165.402,355.467,-78.851,-176.299,8.816,148.688
C03135=1165.405,355.219,-78.817,-176.301,8.812,148.688
C03136=1165.409,354.971,-78.782,-176.303,8.808,148.688
C03137=1165.413,354.723,-78.749,-176.306,8.804,148.687
C03138=1165.418,354.476,-78.714,-176.308,8.801,148.687
C03139=1165.421,354.228,-78.680,-176.311,8.798,148.687
C03140=1165.425,353.980,-78.645,-176.313,8.793,148.686
C03141=1165.429,353.733,-78.612,-176.316,8.790,148.686
C03142=1165.434,353.485,-78.578,-176.318,8.787,148.686
C03143=1165.437,353.237,-78.544,-176.321,8.783,148.686
C03144=1165.441,352.990,-78.510,-176.323,8.779,148.685
C03145=1165.446,352.743,-78.475,-176.325,8.776,148.685
C03146=1165.449,352.494,-78.442,-176.328,8.772,148.685
C03147=1165.454,352.247,-78.407,-176.330,8.768,148.685
C03148=1165.458,352.000,-78.373,-176.332,8.765,148.684
C03149=1165.461,351.751,-78.340,-176.335,8.761,148.684
C03150=1165.466,351.504,-78.305,-176.337,8.757,148.684
C03151=1165.470,351.256,-78.272,-176.339,8.754,148.683
C03152=1165.474,351.009,-78.238,-176.342,8.750,148.683
C03153=1165.478,350.761,-78.204,-176.344,8.747,148.683
C03154=1165.482,350.513,-78.170,-176.347,8.743,148.683
C03155=1165.486,350.266,-78.137,-176.350,8.739,148.682
C03156=1165.490,350.018,-78.102,-176.352,8.736,148.682
C03157=1165.494,349.770,-78.069,-176.354,8.732,148.682
C03158=1165.498,349.523,-78.035,-176.357,8.728,148.682
C03159=1165.502,349.275,-78.001,-176.359,8.725,148.681
C03160=1165.506,349.027,-77.967,-176.361,8.722,148.681
C03161=1165.510,348.780,-77.934,-176.364,8.717,148.681
C03162=1165.514,348.532,-77.900,-176.366,8.714,148.681
C03163=1165.519,348.285,-77.866,-176.369,8.711,148.680
C03164=1165.523,348.037,-77.833,-176.372,8.707,148.680
C03165=1165.526,347.789,-77.799,-176.374,8.703,148.680
C03166=1165.530,347.541,-77.765,-176.376,8.700,148.680
C03167=1165.535,347.294,-77.731,-176.378,8.697,148.679
C03168=1165.539,347.046,-77.698,-176.381,8.692,148.679
C03169=1165.542,346.798,-77.664,-176.383,8.689,148.679
C03170=1165.546,346.551,-77.630,-176.385,8.686,148.679
C03171=1165.550,346.303,-77.597,-176.388,8.682,148.678
C03172=1165.555,346.055,-77.563,-176.391,8.678,148.678
C03173=1165.559,345.808,-77.530,-176.393,8.675,148.678
C03174=1165.563,345.560,-77.496,-176.396,8.671,148.678
C03175=1165.567,345.312,-77.463,-176.398,8.668,148.678
C03176=1165.571,345.064,-77.430,-176.400,8.664,148.677
C03177=1165.575,344.817,-77.396,-176.403,8.661,148.677
C03178=1165.579,344.569,-77.363,-176.406,8.657,148.677
C03179=1165.584,344.321,-77.329,-176.408,8.654,148.677
C03180=1165.588,344.073,-77.296,-176.410,8.650,148.676
C03181=1165.592,343.826,-77.262,-176.413,8.646,148.676
C03182=1165.595,343.578,-77.228,-176.415,8.643,148.676
C03183=1165.599,343.330,-77.195,-176.418,8.640,148.676
C03184=1165.603,343.082,-77.162,-176.420,8.636,148.676
C03185=1165.608,342.835,-77.129,-176.423,8.632,148.675
C03186=1165.612,342.587,-77.096,-176.425,8.629,148.675
C03187=1165.616,342.340,-77.062,-176.427,8.626,148.675
C03188=1165.620,342.092,-77.029,-176.430,8.622,148.675
C03189=1165.624,341.844,-76.996,-176.432,8.618,148.674
C03190=1165.628,341.596,-76.962,-176.435,8.615,148.674
C03191=1165.632,341.349,-76.929,-176.437,8.612,148.674
C03192=1165.636,341.101,-76.896,-176.439,8.608,148.674
C03193=1165.640,340.853,-76.863,-176.442,8.604,148.674
C03194=1165.644,340.605,-76.829,-176.445,8.601,148.673
C03195=1165.648,340.357,-76.796,-176.447,8.598,148.673
C03196=1165.653,340.078,-76.759,-176.450,8.594,148.673
C03197=1165.658,339.799,-76.722,-176.453,8.590,148.673
C03198=1165.662,339.519,-76.684,-176.456,8.586,148.673
C03199=1165.667,339.240,-76.647,-176.458,8.582,148.672
C03200=1165.671,338.991,-76.614,-176.461,8.578,148.672
C03201=1165.676,338.743,-76.581,-176.463,8.575,148.672
C03202=1165.680,338.496,-76.548,-176.466,8.572,148.672
C03203=1165.684,338.248,-76.515,-176.468,8.568,148.671
C03204=1165.688,338.000,-76.482,-176.471,8.564,148.671
C03205=1165.691,337.753,-76.449,-176.473,8.561,148.671
C03206=1165.696,337.505,-76.416,-176.475,8.558,148.671
C03207=1165.700,337.257,-76.383,-176.478,8.555,148.671
C03208=1165.704,337.009,-76.350,-176.481,8.551,148.671
C03209=1165.708,336.761,-76.317,-176.483,8.547,148.670
C03210=1165.712,336.514,-76.284,-176.486,8.544,148.670
C03211=1165.716,336.266,-76.251,-176.488,8.541,148.670
C03212=1165.720,336.018,-76.218,-176.490,8.537,148.670
C03213=1165.724,335.770,-76.186,-176.493,8.533,148.669
C03214=1165.729,335.522,-76.153,-176.496,8.530,148.669
C03215=1165.733,335.275,-76.119,-176.498,8.527,148.669
C03216=1165.736,335.027,-76.087,-176.500,8.524,148.669
C03217=1165.741,334.779,-76.054,-176.503,8.520,148.669
C03218=1165.745,334.531,-76.021,-176.505,8.516,148.669
C03219=1165.749,334.283,-75.988,-176.508,8.513,148.668
C03220=1165.753,334.035,-75.956,-176.510,8.510,148.668
C03221=1165.757,333.788,-75.923,-176.513,8.507,148.668
C03222=1165.761,333.540,-75.890,-176.516,8.503,148.668
C03223=1165.765,333.292,-75.858,-176.518,8.499,148.668
C03224=1165.769,333.044,-75.825,-176.520,8.496,148.668
C03225=1165.773,332.796,-75.793,-176.523,8.493,148.667
C03226=1165.778,332.549,-75.760,-176.525,8.490,148.667
C03227=1165.782,332.301,-75.728,-176.528,8.486,148.667
C03228=1165.786,332.053,-75.695,-176.530,8.482,148.667
C03229=1165.790,331.805,-75.662,-176.533,8.479,148.667
C03230=1165.793,331.557,-75.630,-176.535,8.476,148.666
C03231=1165.798,331.309,-75.597,-176.538,8.473,148.666
C03232=1165.802,331.061,-75.564,-176.541,8.469,148.666
C03233=1165.805,330.814,-75.532,-176.543,8.465,148.666
C03234=1165.811,330.566,-75.499,-176.545,8.462,148.666
C03235=1165.815,330.318,-75.467,-176.548,8.459,148.666
C03236=1165.818,330.070,-75.434,-176.550,8.456,148.666
C03237=1165.823,329.822,-75.402,-176.553,8.452,148.665
C03238=1165.826,329.575,-75.369,-176.555,8.448,148.665
C03239=1165.831,329.326,-75.337,-176.558,8.446,148.665
C03240=1165.836,329.079,-75.305,-176.560,8.442,148.665
C03241=1165.839,328.831,-75.272,-176.563,8.439,148.665
C03242=1165.844,328.583,-75.240,-176.566,8.435,148.665
C03243=1165.847,328.335,-75.207,-176.568,8.432,148.665
C03244=1165.851,328.087,-75.175,-176.571,8.429,148.664
C03245=1165.855,327.839,-75.143,-176.573,8.425,148.664
C03246=1165.860,327.591,-75.111,-176.575,8.422,148.664
C03247=1165.864,327.344,-75.078,-176.578,8.419,148.664
C03248=1165.868,327.096,-75.046,-176.581,8.415,148.664
C03249=1165.872,326.847,-75.014,-176.583,8.412,148.664
C03250=1165.877,326.600,-74.982,-176.586,8.409,148.664
C03251=1165.880,326.352,-74.950,-176.588,8.405,148.663
C03252=1165.885,326.104,-74.917,-176.590,8.402,148.663
C03253=1165.888,325.856,-74.885,-176.593,8.399,148.663
C03254=1165.893,325.608,-74.853,-176.596,8.395,148.663
C03255=1165.897,325.360,-74.821,-176.598,8.392,148.663
C03256=1165.901,325.113,-74.788,-176.601,8.388,148.662
C03257=1165.905,324.865,-74.756,-176.603,8.385,148.662
C03258=1165.910,324.617,-74.724,-176.606,8.382,148.662
C03259=1165.914,324.369,-74.692,-176.608,8.379,148.662
C03260=1165.917,324.121,-74.661,-176.611,8.375,148.662
C03261=1165.922,323.872,-74.628,-176.614,8.372,148.662
C03262=1165.926,323.625,-74.597,-176.616,8.368,148.662
C03263=1165.930,323.377,-74.565,-176.619,8.365,148.662
C03264=1165.934,323.129,-74.532,-176.621,8.362,148.661
C03265=1165.938,322.881,-74.501,-176.623,8.359,148.661
C03266=1165.942,322.634,-74.468,-176.626,8.356,148.661
C03267=1165.946,322.386,-74.436,-176.629,8.352,148.661
C03268=1165.950,322.138,-74.404,-176.631,8.348,148.661
C03269=1165.954,321.890,-74.373,-176.634,8.345,148.661
C03270=1165.959,321.641,-74.341,-176.636,8.342,148.661
C03271=1165.963,321.393,-74.309,-176.638,8.339,148.660
C03272=1165.967,321.146,-74.278,-176.641,8.336,148.660
C03273=1165.972,320.898,-74.245,-176.643,8.333,148.660
C03274=1165.975,320.650,-74.213,-176.647,8.329,148.660
C03275=1165.980,320.402,-74.182,-176.649,8.326,148.660
C03276=1165.983,320.154,-74.150,-176.651,8.322,148.660
C03277=1165.988,319.906,-74.117,-176.654,8.319,148.660
C03278=1165.992,319.658,-74.086,-176.656,8.316,148.660
C03279=1165.996,319.410,-74.054,-176.659,8.313,148.659
C03280=1166.000,319.162,-74.023,-176.661,8.310,148.659
C03281=1166.004,318.914,-73.992,-176.664,8.306,148.659
C03282=1166.009,318.666,-73.959,-176.667,8.303,148.659
C03283=1166.013,318.419,-73.928,-176.669,8.299,148.659
C03284=1166.017,318.171,-73.896,-176.672,8.296,148.659
C03285=1166.021,317.923,-73.865,-176.674,8.293,148.659
C03286=1166.025,317.675,-73.833,-176.677,8.290,148.659
C03287=1166.029,317.426,-73.801,-176.679,8.287,148.659
C03288=1166.034,317.179,-73.769,-176.682,8.283,148.659
C03289=1166.038,316.930,-73.738,-176.684,8.280,148.658
C03290=1166.042,316.683,-73.707,-176.687,8.276,148.658
C03291=1166.046,316.435,-73.675,-176.689,8.273,148.658
C03292=1166.050,316.187,-73.644,-176.692,8.270,148.658
C03293=1166.054,315.939,-73.612,-176.695,8.267,148.658
C03294=1166.058,315.691,-73.580,-176.697,8.264,148.658
C03295=1166.063,315.443,-73.549,-176.700,8.261,148.658
C03296=1166.067,315.195,-73.517,-176.702,8.258,148.658
C03297=1166.071,314.947,-73.486,-176.705,8.254,148.658
C03298=1166.075,314.699,-73.455,-176.707,8.251,148.657
C03299=1166.079,314.451,-73.423,-176.710,8.248,148.657
C03300=1166.085,314.174,-73.389,-176.712,8.244,148.657
C03301=1166.088,313.897,-73.354,-176.716,8.240,148.657
C03302=1166.093,313.620,-73.318,-176.718,8.237,148.657
C03303=1166.098,313.343,-73.283,-176.721,8.233,148.657
C03304=1166.102,313.094,-73.252,-176.724,8.230,148.657
C03305=1166.106,312.847,-73.220,-176.726,8.227,148.657
C03306=1166.110,312.598,-73.189,-176.729,8.223,148.657
C03307=1166.115,312.351,-73.158,-176.731,8.221,148.657
C03308=1166.119,312.102,-73.127,-176.734,8.217,148.656
C03309=1166.123,311.854,-73.096,-176.737,8.214,148.656
C03310=1166.127,311.606,-73.064,-176.739,8.211,148.656
C03311=1166.132,311.358,-73.033,-176.742,8.208,148.656
C03312=1166.136,311.111,-73.002,-176.744,8.204,148.656
C03313=1166.140,310.862,-72.971,-176.747,8.201,148.656
C03314=1166.145,310.614,-72.940,-176.749,8.198,148.656
C03315=1166.148,310.366,-72.908,-176.752,8.195,148.656
C03316=1166.153,310.118,-72.877,-176.754,8.191,148.656
C03317=1166.156,309.870,-72.847,-176.757,8.188,148.656
C03318=1166.160,309.623,-72.815,-176.760,8.185,148.655
C03319=1166.165,309.375,-72.785,-176.762,8.182,148.656
C03320=1166.169,309.126,-72.753,-176.765,8.179,148.655
C03321=1166.173,308.879,-72.722,-176.767,8.176,148.655
C03322=1166.177,308.630,-72.691,-176.770,8.173,148.655
C03323=1166.182,308.382,-72.660,-176.772,8.170,148.655
C03324=1166.187,308.134,-72.629,-176.775,8.166,148.655
C03325=1166.190,307.886,-72.599,-176.777,8.163,148.655
C03326=1166.194,307.639,-72.567,-176.780,8.159,148.655
C03327=1166.199,307.391,-72.536,-176.783,8.156,148.655
C03328=1166.203,307.142,-72.505,-176.785,8.153,148.655
C03329=1166.207,306.894,-72.475,-176.788,8.150,148.655
C03330=1166.211,306.645,-72.443,-176.791,8.147,148.655
C03331=1166.215,306.398,-72.413,-176.793,8.144,148.654
C03332=1166.220,306.150,-72.383,-176.796,8.141,148.654
C03333=1166.224,305.902,-72.351,-176.798,8.137,148.654
C03334=1166.228,305.654,-72.320,-176.801,8.134,148.654
C03335=1166.232,305.406,-72.290,-176.803,8.131,148.654
C03336=1166.237,305.158,-72.259,-176.806,8.128,148.654
C03337=1166.241,304.909,-72.228,-176.808,8.125,148.654
C03338=1166.245,304.662,-72.197,-176.811,8.122,148.654
C03339=1166.249,304.414,-72.167,-176.814,8.119,148.654
C03340=1166.253,304.165,-72.136,-176.816,8.116,148.654
C03341=1166.258,303.917,-72.105,-176.819,8.113,148.654
C03342=1166.262,303.669,-72.074,-176.821,8.109,148.654
C03343=1166.266,303.421,-72.044,-176.824,8.106,148.654
C03344=1166.270,303.173,-72.013,-176.826,8.103,148.654
C03345=1166.275,302.925,-71.982,-176.829,8.099,148.653
C03346=1166.279,302.677,-71.952,-176.832,8.096,148.654
C03347=1166.283,302.429,-71.921,-176.834,8.093,148.653
C03348=1166.288,302.180,-71.891,-176.837,8.090,148.653
C03349=1166.292,301.933,-71.861,-176.839,8.087,148.653
C03350=1166.296,301.685,-71.830,-176.842,8.084,148.653
C03351=1166.300,301.436,-71.799,-176.845,8.081,148.653
C03352=1166.304,301.188,-71.769,-176.847,8.078,148.653
C03353=1166.309,300.940,-71.738,-176.850,8.075,148.653
C03354=1166.313,300.693,-71.708,-176.852,8.071,148.653
C03355=1166.318,300.444,-71.678,-176.855,8.068,148.653
C03356=1166.321,300.196,-71.647,-176.858,8.065,148.653
C03357=1166.325,299.948,-71.616,-176.860,8.062,148.653
C03358=1166.329,299.700,-71.586,-176.863,8.059,148.653
C03359=1166.334,299.452,-71.556,-176.865,8.056,148.653
C03360=1166.338,299.203,-71.525,-176.868,8.053,148.653
C03361=1166.342,298.955,-71.495,-176.870,8.050,148.653
C03362=1166.347,298.707,-71.464,-176.873,8.047,148.652
C03363=1166.351,298.459,-71.435,-176.876,8.044,148.653
C03364=1166.356,298.211,-71.404,-176.878,8.041,148.653
C03365=1166.359,297.963,-71.374,-176.881,8.037,148.652
C03366=1166.364,297.714,-71.343,-176.883,8.034,148.652
C03367=1166.368,297.466,-71.313,-176.886,8.031,148.652
C03368=1166.372,297.219,-71.282,-176.888,8.028,148.652
C03369=1166.376,296.970,-71.253,-176.891,8.025,148.652
C03370=1166.380,296.723,-71.223,-176.894,8.022,148.652
C03371=1166.385,296.474,-71.193,-176.896,8.019,148.652
C03372=1166.389,296.226,-71.163,-176.899,8.016,148.652
C03373=1166.393,295.978,-71.131,-176.902,8.013,148.652
C03374=1166.397,295.729,-71.102,-176.904,8.010,148.652
C03375=1166.402,295.481,-71.071,-176.907,8.007,148.652
C03376=1166.406,295.233,-71.042,-176.909,8.004,148.652
C03377=1166.410,294.986,-71.012,-176.912,8.000,148.652
C03378=1166.415,294.737,-70.981,-176.914,7.997,148.652
C03379=1166.419,294.489,-70.951,-176.917,7.994,148.652
C03380=1166.423,294.241,-70.922,-176.919,7.991,148.652
C03381=1166.428,293.993,-70.891,-176.922,7.988,148.652
C03382=1166.431,293.744,-70.861,-176.925,7.985,148.652
C03383=1166.435,293.496,-70.832,-176.927,7.982,148.652
C03384=1166.440,293.248,-70.801,-176.930,7.979,148.652
C03385=1166.444,293.000,-70.772,-176.933,7.976,148.652
C03386=1166.448,292.752,-70.741,-176.935,7.973,148.652
C03387=1166.453,292.503,-70.711,-176.938,7.970,148.652
C03388=1166.457,292.255,-70.682,-176.941,7.967,148.652
C03389=1166.461,292.008,-70.652,-176.943,7.964,148.652
C03390=1166.465,291.759,-70.622,-176.946,7.961,148.651
C03391=1166.470,291.511,-70.592,-176.948,7.958,148.651
C03392=1166.474,291.263,-70.562,-176.951,7.955,148.652
C03393=1166.478,291.015,-70.533,-176.953,7.951,148.651
C03394=1166.483,290.766,-70.503,-176.956,7.948,148.651
C03395=1166.487,290.519,-70.472,-176.959,7.945,148.651
C03396=1166.491,290.270,-70.443,-176.962,7.942,148.651
C03397=1166.495,290.022,-70.414,-176.964,7.939,148.651
C03398=1166.499,289.774,-70.384,-176.967,7.936,148.651
C03399=1166.504,289.526,-70.353,-176.969,7.933,148.651
C03400=1166.508,289.277,-70.324,-176.972,7.930,148.651
C03401=1166.512,289.029,-70.294,-176.974,7.927,148.651
C03402=1166.517,288.781,-70.265,-176.977,7.925,148.651
C03403=1166.521,288.533,-70.235,-176.979,7.922,148.651
C03404=1166.525,288.258,-70.202,-176.983,7.918,148.651
C03405=1166.530,287.983,-70.170,-176.985,7.915,148.651
C03406=1166.535,287.708,-70.136,-176.988,7.911,148.651
C03407=1166.540,287.432,-70.104,-176.991,7.908,148.651
C03408=1166.544,287.184,-70.074,-176.994,7.905,148.651
C03409=1166.548,286.936,-70.045,-176.997,7.902,148.651
C03410=1166.553,286.688,-70.016,-176.999,7.899,148.651
C03411=1166.557,286.440,-69.986,-177.002,7.896,148.651
C03412=1166.561,286.192,-69.957,-177.004,7.893,148.651
C03413=1166.565,285.944,-69.927,-177.007,7.890,148.651
C03414=1166.570,285.696,-69.897,-177.010,7.887,148.651
C03415=1166.574,285.448,-69.868,-177.012,7.884,148.651
C03416=1166.578,285.199,-69.839,-177.015,7.881,148.651
C03417=1166.582,284.950,-69.809,-177.017,7.878,148.651
C03418=1166.587,284.702,-69.780,-177.020,7.876,148.651
C03419=1166.591,284.454,-69.751,-177.022,7.872,148.651
C03420=1166.595,284.206,-69.721,-177.025,7.869,148.651
C03421=1166.600,283.958,-69.691,-177.028,7.866,148.651
C03422=1166.605,283.709,-69.662,-177.030,7.863,148.651
C03423=1166.609,283.461,-69.633,-177.033,7.860,148.651
C03424=1166.612,283.213,-69.604,-177.035,7.857,148.651
C03425=1166.616,282.965,-69.574,-177.038,7.854,148.651
C03426=1166.621,282.717,-69.545,-177.041,7.851,148.651
C03427=1166.626,282.469,-69.516,-177.044,7.848,148.651
C03428=1166.630,282.220,-69.487,-177.046,7.845,148.651
C03429=1166.634,281.972,-69.457,-177.049,7.842,148.651
C03430=1166.638,281.724,-69.428,-177.051,7.839,148.651
C03431=1166.642,281.475,-69.399,-177.054,7.837,148.651
C03432=1166.647,281.227,-69.370,-177.056,7.834,148.651
C03433=1166.652,280.979,-69.341,-177.059,7.831,148.651
C03434=1166.656,280.731,-69.311,-177.062,7.828,148.651
C03435=1166.660,280.482,-69.282,-177.064,7.825,148.651
C03436=1166.665,280.234,-69.253,-177.067,7.822,148.651
C03437=1166.669,279.985,-69.224,-177.070,7.819,148.651
C03438=1166.673,279.738,-69.195,-177.072,7.816,148.651
C03439=1166.677,279.489,-69.166,-177.075,7.813,148.651
C03440=1166.681,279.241,-69.137,-177.078,7.810,148.651
C03441=1166.686,278.993,-69.108,-177.080,7.807,148.651
C03442=1166.690,278.744,-69.079,-177.083,7.804,148.651
C03443=1166.695,278.496,-69.050,-177.085,7.801,148.651
C03444=1166.698,278.248,-69.021,-177.088,7.798,148.651
C03445=1166.703,277.999,-68.992,-177.091,7.795,148.651
C03446=1166.707,277.751,-68.963,-177.093,7.793,148.651
C03447=1166.712,277.503,-68.934,-177.096,7.790,148.651
C03448=1166.716,277.255,-68.905,-177.099,7.787,148.651
C03449=1166.720,277.006,-68.877,-177.101,7.783,148.651
C03450=1166.724,276.758,-68.847,-177.104,7.780,148.651
C03451=1166.729,276.510,-68.819,-177.107,7.777,148.651
C03452=1166.733,276.262,-68.790,-177.109,7.774,148.651
C03453=1166.737,276.013,-68.761,-177.112,7.772,148.652
C03454=1166.742,275.765,-68.732,-177.114,7.769,148.652
C03455=1166.746,275.516,-68.703,-177.117,7.766,148.652
C03456=1166.750,275.268,-68.675,-177.120,7.763,148.652
C03457=1166.755,275.020,-68.646,-177.122,7.760,148.651
C03458=1166.759,274.772,-68.617,-177.125,7.757,148.652
C03459=1166.763,274.523,-68.589,-177.128,7.754,148.652
C03460=1166.767,274.275,-68.559,-177.130,7.751,148.652
C03461=1166.772,274.027,-68.531,-177.133,7.749,148.652
C03462=1166.776,273.778,-68.503,-177.135,7.746,148.652
C03463=1166.780,273.530,-68.473,-177.138,7.743,148.652
C03464=1166.785,273.282,-68.445,-177.141,7.740,148.652
C03465=1166.789,273.033,-68.417,-177.144,7.737,148.652
C03466=1166.794,272.786,-68.388,-177.146,7.734,148.652
C03467=1166.798,272.537,-68.359,-177.149,7.731,148.652
C03468=1166.802,272.288,-68.331,-177.151,7.728,148.652
C03469=1166.807,272.041,-68.302,-177.153,7.726,148.652
C03470=1166.811,271.792,-68.273,-177.156,7.723,148.652
C03471=1166.815,271.543,-68.245,-177.159,7.720,148.652
C03472=1166.820,271.295,-68.216,-177.162,7.717,148.652
C03473=1166.824,271.047,-68.188,-177.165,7.714,148.652
C03474=1166.829,270.799,-68.159,-177.167,7.711,148.652
C03475=1166.832,270.550,-68.131,-177.170,7.708,148.652
C03476=1166.837,270.301,-68.102,-177.172,7.706,148.652
C03477=1166.841,270.054,-68.074,-177.175,7.703,148.652
C03478=1166.846,269.805,-68.046,-177.178,7.700,148.652
C03479=1166.850,269.557,-68.017,-177.180,7.697,148.652
C03480=1166.854,269.308,-67.989,-177.183,7.694,148.652
C03481=1166.859,269.061,-67.961,-177.186,7.691,148.653
C03482=1166.863,268.812,-67.932,-177.189,7.688,148.653
C03483=1166.867,268.563,-67.904,-177.191,7.686,148.653
C03484=1166.872,268.315,-67.875,-177.194,7.683,148.653
C03485=1166.876,268.066,-67.847,-177.196,7.680,148.653
C03486=1166.881,267.818,-67.819,-177.199,7.677,148.653
C03487=1166.885,267.570,-67.791,-177.201,7.674,148.653
C03488=1166.890,267.321,-67.762,-177.204,7.671,148.653
C03489=1166.893,267.073,-67.734,-177.206,7.669,148.653
C03490=1166.898,266.825,-67.707,-177.209,7.666,148.653
C03491=1166.902,266.576,-67.678,-177.212,7.663,148.653
C03492=1166.907,266.328,-67.650,-177.215,7.660,148.653
C03493=1166.911,266.079,-67.621,-177.217,7.657,148.653
C03494=1166.915,265.831,-67.594,-177.220,7.654,148.653
C03495=1166.919,265.583,-67.565,-177.222,7.652,148.653
C03496=1166.924,265.335,-67.537,-177.225,7.649,148.653
C03497=1166.928,265.086,-67.509,-177.228,7.646,148.653
C03498=1166.933,264.838,-67.480,-177.231,7.643,148.653
C03499=1166.937,264.589,-67.452,-177.233,7.640,148.653
C03500=1166.941,264.341,-67.425,-177.236,7.637,148.653
C03501=1166.946,264.093,-67.396,-177.238,7.635,148.654
C03502=1166.950,263.844,-67.369,-177.241,7.632,148.654
C03503=1166.955,263.596,-67.341,-177.244,7.629,148.654
C03504=1166.959,263.347,-67.312,-177.247,7.626,148.654
C03505=1166.963,263.099,-67.284,-177.249,7.623,148.654
C03506=1166.967,262.851,-67.256,-177.251,7.621,148.654
C03507=1166.972,262.602,-67.229,-177.254,7.618,148.654
C03508=1166.976,262.330,-67.198,-177.257,7.615,148.654
C03509=1166.981,262.056,-67.167,-177.261,7.611,148.654
C03510=1166.986,261.783,-67.137,-177.264,7.609,148.654
C03511=1166.991,261.510,-67.106,-177.266,7.606,148.654
C03512=1166.996,261.261,-67.078,-177.269,7.603,148.654
C03513=1167.000,261.013,-67.050,-177.272,7.600,148.654
C03514=1167.004,260.764,-67.022,-177.274,7.598,148.654
C03515=1167.008,260.517,-66.994,-177.277,7.595,148.655
C03516=1167.013,260.268,-66.967,-177.279,7.592,148.655
C03517=1167.017,260.019,-66.939,-177.282,7.589,148.655
C03518=1167.022,259.771,-66.912,-177.285,7.586,148.655
C03519=1167.026,259.523,-66.884,-177.287,7.584,148.655
C03520=1167.030,259.274,-66.856,-177.290,7.581,148.655
C03521=1167.035,259.026,-66.829,-177.293,7.578,148.655
C03522=1167.040,258.778,-66.800,-177.296,7.575,148.655
C03523=1167.044,258.528,-66.773,-177.298,7.573,148.655
C03524=1167.048,258.280,-66.745,-177.301,7.570,148.655
C03525=1167.052,258.033,-66.717,-177.304,7.567,148.655
C03526=1167.057,257.783,-66.690,-177.306,7.564,148.655
C03527=1167.061,257.536,-66.662,-177.309,7.561,148.656
C03528=1167.066,257.287,-66.635,-177.311,7.559,148.656
C03529=1167.069,257.038,-66.607,-177.314,7.556,148.656
C03530=1167.074,256.790,-66.580,-177.317,7.553,148.656
C03531=1167.078,256.542,-66.552,-177.320,7.550,148.656
C03532=1167.083,256.293,-66.524,-177.322,7.548,148.656
C03533=1167.088,256.044,-66.497,-177.325,7.545,148.656
C03534=1167.092,255.796,-66.469,-177.328,7.542,148.656
C03535=1167.096,255.547,-66.442,-177.330,7.539,148.656
C03536=1167.101,255.299,-66.414,-177.333,7.537,148.656
C03537=1167.105,255.051,-66.387,-177.335,7.534,148.656
C03538=1167.110,254.802,-66.360,-177.338,7.531,148.656
C03539=1167.114,254.554,-66.332,-177.341,7.528,148.657
C03540=1167.118,254.305,-66.305,-177.344,7.525,148.657
C03541=1167.123,254.057,-66.277,-177.346,7.523,148.657
C03542=1167.127,253.809,-66.250,-177.349,7.521,148.657
C03543=1167.131,253.559,-66.222,-177.352,7.518,148.657
C03544=1167.136,253.311,-66.195,-177.355,7.515,148.657
C03545=1167.140,253.063,-66.168,-177.357,7.513,148.657
C03546=1167.144,252.815,-66.141,-177.360,7.510,148.657
C03547=1167.148,252.566,-66.114,-177.362,7.507,148.657
C03548=1167.153,252.318,-66.086,-177.364,7.505,148.657
C03549=1167.157,252.069,-66.059,-177.368,7.502,148.658
C03550=1167.162,251.821,-66.032,-177.370,7.499,148.658
C03551=1167.167,251.572,-66.005,-177.373,7.496,148.658
C03552=1167.171,251.323,-65.977,-177.375,7.494,148.658
C03553=1167.175,251.075,-65.949,-177.378,7.491,148.658
C03554=1167.180,250.827,-65.922,-177.381,7.488,148.658
C03555=1167.184,250.578,-65.895,-177.384,7.485,148.658
C03556=1167.188,250.330,-65.869,-177.386,7.483,148.658
C03557=1167.193,250.082,-65.842,-177.389,7.480,148.659
C03558=1167.197,249.832,-65.814,-177.392,7.477,148.659
C03559=1167.202,249.584,-65.787,-177.395,7.474,148.659
C03560=1167.206,249.335,-65.760,-177.397,7.472,148.659
C03561=1167.211,249.088,-65.733,-177.400,7.469,148.659
C03562=1167.215,248.839,-65.706,-177.403,7.467,148.659
C03563=1167.219,248.591,-65.679,-177.405,7.464,148.659
C03564=1167.224,248.342,-65.652,-177.408,7.461,148.659
C03565=1167.228,248.093,-65.624,-177.410,7.459,148.659
C03566=1167.233,247.845,-65.597,-177.413,7.456,148.659
C03567=1167.236,247.597,-65.571,-177.416,7.454,148.660
C03568=1167.241,247.348,-65.544,-177.419,7.451,148.660
C03569=1167.246,247.100,-65.517,-177.421,7.448,148.660
C03570=1167.250,246.851,-65.490,-177.424,7.446,148.660
C03571=1167.254,246.603,-65.463,-177.426,7.443,148.660
C03572=1167.259,246.354,-65.436,-177.430,7.440,148.660
C03573=1167.264,246.105,-65.410,-177.432,7.438,148.660
C03574=1167.269,245.857,-65.383,-177.435,7.435,148.660
C03575=1167.272,245.608,-65.356,-177.437,7.432,148.661
C03576=1167.277,245.359,-65.329,-177.440,7.429,148.661
C03577=1167.281,245.111,-65.302,-177.443,7.427,148.661
C03578=1167.285,244.863,-65.275,-177.445,7.424,148.661
C03579=1167.290,244.614,-65.248,-177.448,7.421,148.661
C03580=1167.295,244.366,-65.221,-177.450,7.419,148.661
C03581=1167.299,244.117,-65.196,-177.454,7.417,148.661
C03582=1167.303,243.868,-65.168,-177.456,7.414,148.661
C03583=1167.307,243.620,-65.142,-177.459,7.412,148.662
C03584=1167.312,243.372,-65.115,-177.461,7.409,148.662
C03585=1167.317,243.123,-65.088,-177.465,7.406,148.662
C03586=1167.321,242.874,-65.062,-177.467,7.404,148.662
C03587=1167.326,242.626,-65.035,-177.469,7.401,148.662
C03588=1167.330,242.377,-65.008,-177.472,7.398,148.662
C03589=1167.334,242.129,-64.982,-177.475,7.396,148.663
C03590=1167.339,241.880,-64.955,-177.478,7.393,148.663
C03591=1167.343,241.632,-64.929,-177.480,7.390,148.663
C03592=1167.348,241.383,-64.902,-177.483,7.388,148.663
C03593=1167.352,241.135,-64.876,-177.486,7.386,148.663
C03594=1167.357,240.886,-64.849,-177.489,7.383,148.663
C03595=1167.360,240.638,-64.822,-177.491,7.380,148.663
C03596=1167.365,240.389,-64.796,-177.494,7.378,148.663
C03597=1167.369,240.141,-64.770,-177.497,7.375,148.664
C03598=1167.374,239.892,-64.743,-177.499,7.373,148.664
C03599=1167.378,239.643,-64.717,-177.502,7.370,148.664
C03600=1167.383,239.395,-64.690,-177.505,7.367,148.664
C03601=1167.387,239.146,-64.664,-177.507,7.365,148.664
C03602=1167.392,238.898,-64.637,-177.510,7.362,148.664
C03603=1167.396,238.649,-64.611,-177.513,7.359,148.664
C03604=1167.401,238.400,-64.584,-177.515,7.357,148.665
C03605=1167.405,238.152,-64.559,-177.518,7.354,148.665
C03606=1167.410,237.904,-64.532,-177.521,7.351,148.665
C03607=1167.414,237.655,-64.506,-177.523,7.350,148.665
C03608=1167.419,237.406,-64.479,-177.526,7.347,148.665
C03609=1167.423,237.158,-64.453,-177.528,7.345,148.665
C03610=1167.427,236.909,-64.427,-177.531,7.342,148.665
C03611=1167.432,236.660,-64.400,-177.534,7.339,148.666
C03612=1167.436,236.389,-64.372,-177.537,7.336,148.666
C03613=1167.442,236.117,-64.343,-177.540,7.333,148.666
C03614=1167.446,235.845,-64.314,-177.543,7.330,148.666
C03615=1167.452,235.573,-64.285,-177.546,7.328,148.666
C03616=1167.456,235.325,-64.259,-177.549,7.326,148.666
C03617=1167.460,235.077,-64.234,-177.551,7.323,148.667
C03618=1167.465,234.828,-64.207,-177.554,7.321,148.667
C03619=1167.469,234.580,-64.181,-177.557,7.318,148.667
C03620=1167.474,234.331,-64.155,-177.560,7.315,148.667
C03621=1167.479,234.082,-64.129,-177.562,7.313,148.667
C03622=1167.482,233.834,-64.102,-177.565,7.310,148.667
C03623=1167.487,233.585,-64.077,-177.567,7.308,148.668
C03624=1167.491,233.337,-64.051,-177.570,7.306,148.668
C03625=1167.496,233.088,-64.024,-177.573,7.303,148.668
C03626=1167.500,232.839,-63.998,-177.575,7.301,148.668
C03627=1167.505,232.591,-63.973,-177.579,7.298,148.668
C03628=1167.509,232.342,-63.947,-177.581,7.296,148.668
C03629=1167.514,232.094,-63.920,-177.584,7.293,148.669
C03630=1167.518,231.845,-63.894,-177.587,7.290,148.669
C03631=1167.523,231.596,-63.869,-177.589,7.288,148.669
C03632=1167.527,231.348,-63.843,-177.592,7.285,148.669
C03633=1167.532,231.099,-63.817,-177.594,7.283,148.669
C03634=1167.537,230.850,-63.791,-177.597,7.280,148.669
C03635=1167.540,230.602,-63.765,-177.600,7.278,148.670
C03636=1167.545,230.353,-63.739,-177.603,7.276,148.670
C03637=1167.550,230.105,-63.714,-177.605,7.273,148.670
C03638=1167.554,229.856,-63.687,-177.608,7.271,148.670
C03639=1167.559,229.607,-63.661,-177.611,7.268,148.670
C03640=1167.563,229.359,-63.636,-177.614,7.265,148.670
C03641=1167.568,229.110,-63.610,-177.616,7.263,148.671
C03642=1167.572,228.862,-63.585,-177.619,7.260,148.671
C03643=1167.576,228.613,-63.559,-177.622,7.258,148.671
C03644=1167.580,228.364,-63.533,-177.624,7.256,148.671
C03645=1167.586,228.116,-63.507,-177.627,7.253,148.671
C03646=1167.590,227.867,-63.481,-177.630,7.251,148.672
C03647=1167.594,227.618,-63.456,-177.633,7.248,148.672
C03648=1167.599,227.370,-63.430,-177.635,7.246,148.672
C03649=1167.603,227.121,-63.404,-177.638,7.243,148.672
C03650=1167.608,226.872,-63.379,-177.640,7.241,148.672
C03651=1167.612,226.623,-63.353,-177.643,7.238,148.673
C03652=1167.617,226.375,-63.328,-177.646,7.236,148.673
C03653=1167.621,226.127,-63.302,-177.649,7.234,148.673
C03654=1167.625,225.878,-63.276,-177.651,7.232,148.673
C03655=1167.630,225.630,-63.251,-177.654,7.229,148.673
C03656=1167.635,225.380,-63.226,-177.656,7.227,148.673
